// TIA Portal V18 program export: 0 tag tables, 0 data types, 8 data blocks, 19 code blocks (in call order from the OBs), 10 instance data blocks

DATA_BLOCK "settingsShift"   // DB23
{ S7_Optimized_Access := 'TRUE' }
VERSION : 0.1
// stored: AutoNumber false, DBAccessibleFromOPCUA true, DBAccessibleFromWebserver true, IsOnlyStoredInLoadMemory false, IsRetainMemResEnabled true, IsWriteProtectedInAS false, MemoryReserve 1000, RetainMemoryReserve 1000
   VAR RETAIN
      "1" { ExternalVisible := 'False'; S7_SetPoint := 'True'} : "UDT_settingsShift";
      "2" { ExternalVisible := 'False'; S7_SetPoint := 'True'} : "UDT_settingsShift";
      "3" { ExternalVisible := 'False'; S7_SetPoint := 'True'} : "UDT_settingsShift";
   END_VAR
BEGIN
END_DATA_BLOCK

DATA_BLOCK "settingsSirene"   // DB25
{ S7_Optimized_Access := 'TRUE' }
VERSION : 0.1
// stored: AutoNumber false, DBAccessibleFromOPCUA true, DBAccessibleFromWebserver true, IsOnlyStoredInLoadMemory false, IsRetainMemResEnabled true, IsWriteProtectedInAS false, MemoryReserve 100, RetainMemoryReserve 100
   VAR RETAIN
      green { S7_SetPoint := 'True'} : "UDT_settingsSirene";
      yellow { S7_SetPoint := 'True'} : "UDT_settingsSirene";
      red { S7_SetPoint := 'True'} : "UDT_settingsSirene";
   END_VAR
BEGIN
END_DATA_BLOCK

DATA_BLOCK "gDb_AndonBoxConfig"   // DB17
{ S7_Optimized_Access := 'TRUE' }
VERSION : 0.1
// stored: AutoNumber true, DBAccessibleFromOPCUA true, DBAccessibleFromWebserver true, IsOnlyStoredInLoadMemory false, IsRetainMemResEnabled false, IsWriteProtectedInAS false, MemoryReserve 100
   VAR RETAIN
      flashingPeriod : Time := T#200ms;
      EnableAndon1 : Bool := true;
      EnableAndon2 : Bool := true;
      EnableAndon3 : Bool := true;
      EnableAndon4 : Bool := true;
      EnableAndon5 : Bool := true;
      EnableAndon6 : Bool := true;
      EnableAndon7 : Bool := true;
      EnableAndon8 : Bool;
      EnableAndon9 : Bool;
      EnableAndon10 : Bool;
   END_VAR
BEGIN
END_DATA_BLOCK

DATA_BLOCK "gDb_LED_state"   // DB9
{ S7_Optimized_Access := 'TRUE' }
VERSION : 0.1
// stored: AutoNumber true, DBAccessibleFromOPCUA true, DBAccessibleFromWebserver true, IsOnlyStoredInLoadMemory false, IsRetainMemResEnabled false, IsWriteProtectedInAS false, MemoryReserve 100
   VAR RETAIN
      green : Bool;
      yellow : Bool;
      red : Bool;
   END_VAR
BEGIN
END_DATA_BLOCK

DATA_BLOCK "gDb_IO"   // DB20
{ S7_Optimized_Access := 'TRUE' }
VERSION : 0.1
// stored: AutoNumber true, DBAccessibleFromOPCUA true, DBAccessibleFromWebserver true, IsOnlyStoredInLoadMemory false, IsRetainMemResEnabled false, IsWriteProtectedInAS false, MemoryReserve 100
   VAR
      Andon1 : "UDT_andonIO";
      Andon2 : "UDT_andonIO";
      Andon3 : "UDT_andonIO";
      Andon4 : "UDT_andonIO";
      Andon5 : "UDT_andonIO";
      Andon6 : "UDT_andonIO";
      Andon7 : "UDT_andonIO";
      Andon8 : "UDT_andonIO";
      Andon9 : "UDT_andonIO";
      Andon10 : "UDT_andonIO";
      Sirene { S7_SetPoint := 'True'} : "UDT_sireneIO";
      SignalColumn { S7_SetPoint := 'True'} : "UDT_signalColumn";
      NokButton1 { S7_SetPoint := 'True'} : "UDT_nokButtonIO";
      NokButton2 { S7_SetPoint := 'True'} : "UDT_nokButtonIO";
      I_PartProduced { S7_SetPoint := 'True'} : Bool;
   END_VAR
BEGIN
END_DATA_BLOCK

DATA_BLOCK "gdb_nokButton"   // DB14
{ S7_Optimized_Access := 'TRUE' }
VERSION : 0.1
// stored: AutoNumber true, DBAccessibleFromOPCUA true, DBAccessibleFromWebserver true, IsOnlyStoredInLoadMemory false, IsRetainMemResEnabled false, IsWriteProtectedInAS false, MemoryReserve 100
   VAR
      ButtonQue : Int;
      nokPart : Bool;
   END_VAR
BEGIN
END_DATA_BLOCK

DATA_BLOCK "gdb_Sirene"   // DB13
{ S7_Optimized_Access := 'TRUE' }
VERSION : 0.1
// stored: AutoNumber true, DBAccessibleFromOPCUA true, DBAccessibleFromWebserver true, IsOnlyStoredInLoadMemory false, IsRetainMemResEnabled false, IsWriteProtectedInAS false, MemoryReserve 100
   VAR
      greenTrigger : Bool;
      yellowTrigger : Bool;
      redTrigger : Bool;
   END_VAR
BEGIN
END_DATA_BLOCK

DATA_BLOCK "webData"   // DB8
{ S7_Optimized_Access := 'TRUE' }
VERSION : 0.1
// stored: AutoNumber true, DBAccessibleFromOPCUA true, DBAccessibleFromWebserver true, IsOnlyStoredInLoadMemory false, IsRetainMemResEnabled false, IsWriteProtectedInAS false, MemoryReserve 0
   VAR
      lineName { ExternalAccessible := 'False'; ExternalVisible := 'False'; ExternalWritable := 'False'} : WString := WSTRING#'L14';
      andon1Text { ExternalAccessible := 'False'; ExternalVisible := 'False'; ExternalWritable := 'False'} : WString := WSTRING#'Andon1';
      andon2Text { ExternalAccessible := 'False'; ExternalVisible := 'False'; ExternalWritable := 'False'} : WString := WSTRING#'Andon2';
      andon3Text { ExternalAccessible := 'False'; ExternalVisible := 'False'; ExternalWritable := 'False'} : WString := WSTRING#'Andon3';
      andon4Text { ExternalAccessible := 'False'; ExternalVisible := 'False'; ExternalWritable := 'False'} : WString := WSTRING#'Andon4';
      andon5Text { ExternalAccessible := 'False'; ExternalVisible := 'False'; ExternalWritable := 'False'} : WString := WSTRING#'Andon5';
      andon6Text { ExternalAccessible := 'False'; ExternalVisible := 'False'; ExternalWritable := 'False'} : WString := WSTRING#'Andon6';
      andon7Text { ExternalAccessible := 'False'; ExternalVisible := 'False'; ExternalWritable := 'False'} : WString := WSTRING#'Andon7';
      andon8Text { ExternalAccessible := 'False'; ExternalVisible := 'False'; ExternalWritable := 'False'} : WString := WSTRING#'Andon8';
      andon9Text { ExternalAccessible := 'False'; ExternalVisible := 'False'; ExternalWritable := 'False'} : WString := WSTRING#'Andon9';
      andon10Text { ExternalAccessible := 'False'; ExternalVisible := 'False'; ExternalWritable := 'False'} : WString := WSTRING#'Andon10';
      actualValues { ExternalAccessible := 'False'; ExternalVisible := 'False'; ExternalWritable := 'False'} : "UDT_actualValues";
      andon1state { ExternalAccessible := 'False'; ExternalVisible := 'False'; ExternalWritable := 'False'} : Int;
      andon2state { ExternalAccessible := 'False'; ExternalVisible := 'False'; ExternalWritable := 'False'} : Int;
      andon3state { ExternalAccessible := 'False'; ExternalVisible := 'False'; ExternalWritable := 'False'} : Int;
      andon4state { ExternalAccessible := 'False'; ExternalVisible := 'False'; ExternalWritable := 'False'} : Int;
      andon5state { ExternalAccessible := 'False'; ExternalVisible := 'False'; ExternalWritable := 'False'} : Int;
      andon6state { ExternalAccessible := 'False'; ExternalVisible := 'False'; ExternalWritable := 'False'} : Int;
      andon7state { ExternalAccessible := 'False'; ExternalVisible := 'False'; ExternalWritable := 'False'} : Int;
      andon8state { ExternalAccessible := 'False'; ExternalVisible := 'False'; ExternalWritable := 'False'} : Int;
      andon9state { ExternalAccessible := 'False'; ExternalVisible := 'False'; ExternalWritable := 'False'} : Int;
      andon10state { ExternalAccessible := 'False'; ExternalVisible := 'False'; ExternalWritable := 'False'} : Int;
   END_VAR
BEGIN
END_DATA_BLOCK

ORGANIZATION_BLOCK "Main"   // OB1, FBD, ProgramCycle
TITLE = "Main Program Sweep (Cycle)"
{ S7_Optimized_Access := 'TRUE' }
// stored: SetENOAutomatically false
   VAR_INPUT
      Initial_Call : Bool;   // Initial call of this OB
      Remanence : Bool;   // =True, if remanent data are available
   END_VAR
   VAR_TEMP
      RET_VAL : Int;
      locTime : DTL;
   END_VAR
BEGIN

REGION Network 1: Inputs
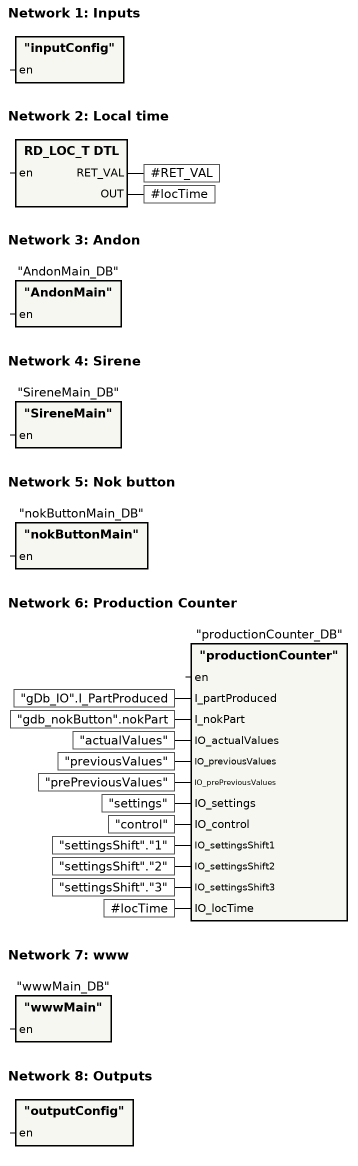
   "inputConfig"();
END_REGION

REGION Network 2: Local time
   #RET_VAL := RD_LOC_T(OUT => #locTime);
END_REGION

REGION Network 3: Andon
   "AndonMain_DB"();   // "AndonMain"
END_REGION

REGION Network 4: Sirene
   "SireneMain_DB"();   // "SireneMain"
END_REGION

REGION Network 5: Nok button
   "nokButtonMain_DB"();   // "nokButtonMain"
END_REGION

REGION Network 6: Production Counter
   "productionCounter_DB"(I_partProduced := "gDb_IO".I_PartProduced,   // "productionCounter"
                          I_nokPart := "gdb_nokButton".nokPart,
                          IO_actualValues := "actualValues",
                          IO_previousValues := "previousValues",
                          IO_prePreviousValues := "prePreviousValues",
                          IO_settings := "settings",
                          IO_control := "control",
                          IO_settingsShift1 := "settingsShift"."1",
                          IO_settingsShift2 := "settingsShift"."2",
                          IO_settingsShift3 := "settingsShift"."3",
                          IO_locTime := #locTime);
END_REGION

REGION Network 7: www
   "wwwMain_DB"();   // "wwwMain"
END_REGION

REGION Network 8: Outputs
   "outputConfig"();
END_REGION
END_ORGANIZATION_BLOCK

FUNCTION "inputConfig" : Void
{ S7_Optimized_Access := 'TRUE' }
VERSION : 0.1

BEGIN
	(*
	//Andon1
	"gDb_IO".Andon1.I_greenBtn := "Andon1_greenBtn";
	"gDb_IO".Andon1.I_yellowBtn := "Andon1_yellowBtn";
	"gDb_IO".Andon1.I_redBtn := "Andon1_redBtn";
	//Andon2
	"gDb_IO".Andon2.I_greenBtn := "Andon2_greenBtn";
	"gDb_IO".Andon2.I_yellowBtn := "Andon2_yellowBtn";
	"gDb_IO".Andon2.I_redBtn := "Andon2_redBtn";
	//Andon7
	"gDb_IO".Andon3.I_greenBtn := "Andon3_greenBtn";
	"gDb_IO".Andon3.I_yellowBtn := "Andon3_yellowBtn";
	"gDb_IO".Andon3.I_redBtn := "Andon3_redBtn";
	//Andon4
	"gDb_IO".Andon4.I_greenBtn := "Andon4_greenBtn";
	"gDb_IO".Andon4.I_yellowBtn := "Andon4_yellowBtn";
	"gDb_IO".Andon4.I_redBtn := "Andon4_redBtn";
	//Andon6
	"gDb_IO".Andon5.I_greenBtn := "Andon5_greenBtn";
	"gDb_IO".Andon5.I_yellowBtn := "Andon5_yellowBtn";
	"gDb_IO".Andon5.I_redBtn := "Andon5_redBtn";
	//Andon6
	"gDb_IO".Andon6.I_greenBtn := "Andon6_greenBtn";
	"gDb_IO".Andon6.I_yellowBtn := "Andon6_yellowBtn";
	"gDb_IO".Andon6.I_redBtn := "Andon6_redBtn";
	//Andon7
	"gDb_IO".Andon7.I_greenBtn := "Andon7_greenBtn";
	"gDb_IO".Andon7.I_yellowBtn := "Andon7_yellowBtn";
	"gDb_IO".Andon7.I_redBtn := "Andon7_redBtn";
	//Andon8
	"gDb_IO".Andon8.I_greenBtn := "Andon8_greenBtn";
	"gDb_IO".Andon8.I_yellowBtn := "Andon8_yellowBtn";
	"gDb_IO".Andon8.I_redBtn := "Andon8_redBtn";
	//Andon9
	"gDb_IO".Andon9.I_greenBtn := "Andon9_greenBtn";
	"gDb_IO".Andon9.I_yellowBtn := "Andon9_yellowBtn";
	"gDb_IO".Andon9.I_redBtn := "Andon9_redBtn";
	*)
END_FUNCTION

FUNCTION_BLOCK "AndonMain"   // FB1, FBD
{ S7_Optimized_Access := 'TRUE' }
VERSION : 0.1
// stored: AutoNumber true, IsIECCheckEnabled false, IsRetainMemResEnabled false, MemoryReserve 100, SetENOAutomatically false, UDAEnableTagReadback false
   VAR
      fpBit_greenTrigger : Bool;
      AndonBoxASi_v2_Instance_8 { S7_SetPoint := 'True'} : "AndonBoxASi";
      AndonBoxASi_v2_Instance_9 { S7_SetPoint := 'True'} : "AndonBoxASi";
      AndonBoxASi_v2_Instance1 { S7_SetPoint := 'True'} : "AndonBoxASi";
      AndonBoxASi_v2_Instance2 { S7_SetPoint := 'True'} : "AndonBoxASi";
      AndonBoxASi_v2_Instance3 { S7_SetPoint := 'True'} : "AndonBoxASi";
      AndonBoxASi_v2_Instance4 { S7_SetPoint := 'True'} : "AndonBoxASi";
      AndonBoxASi_v2_Instance5 { S7_SetPoint := 'True'} : "AndonBoxASi";
      AndonBoxASi_v2_Instance6 { S7_SetPoint := 'True'} : "AndonBoxASi";
      AndonBoxASi_v2_Instance7 { S7_SetPoint := 'True'} : "AndonBoxASi";
      AndonBoxASi_v2_Instance10 { S7_SetPoint := 'True'} : "AndonBoxASi";
   END_VAR
   VAR_TEMP   // added for the SCL form of the ladder/FBD networks
      _w1 : Bool;
      _w2 : Bool;
   END_VAR
BEGIN

REGION Network 1: Green trigger
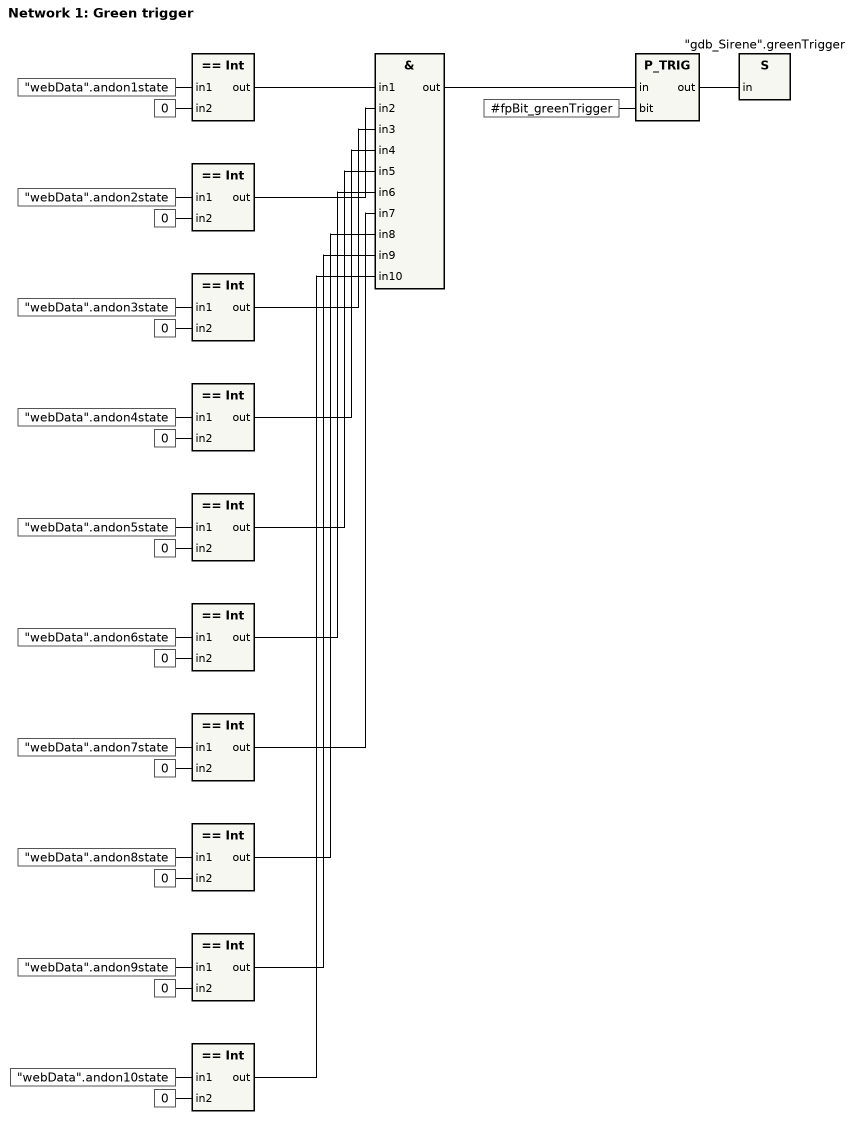
   #_w1 := ("webData".andon1state = 0) AND ("webData".andon2state = 0) AND ("webData".andon3state = 0) AND ("webData".andon4state = 0) AND ("webData".andon5state = 0) AND ("webData".andon6state = 0) AND ("webData".andon7state = 0) AND ("webData".andon8state = 0) AND ("webData".andon9state = 0) AND ("webData".andon10state = 0);
   #_w2 := #_w1 AND NOT #fpBit_greenTrigger;   // rising edge
   #fpBit_greenTrigger := #_w1;
   IF #_w2 THEN "gdb_Sirene".greenTrigger := TRUE; END_IF;
END_REGION

REGION Network 2: Andon1
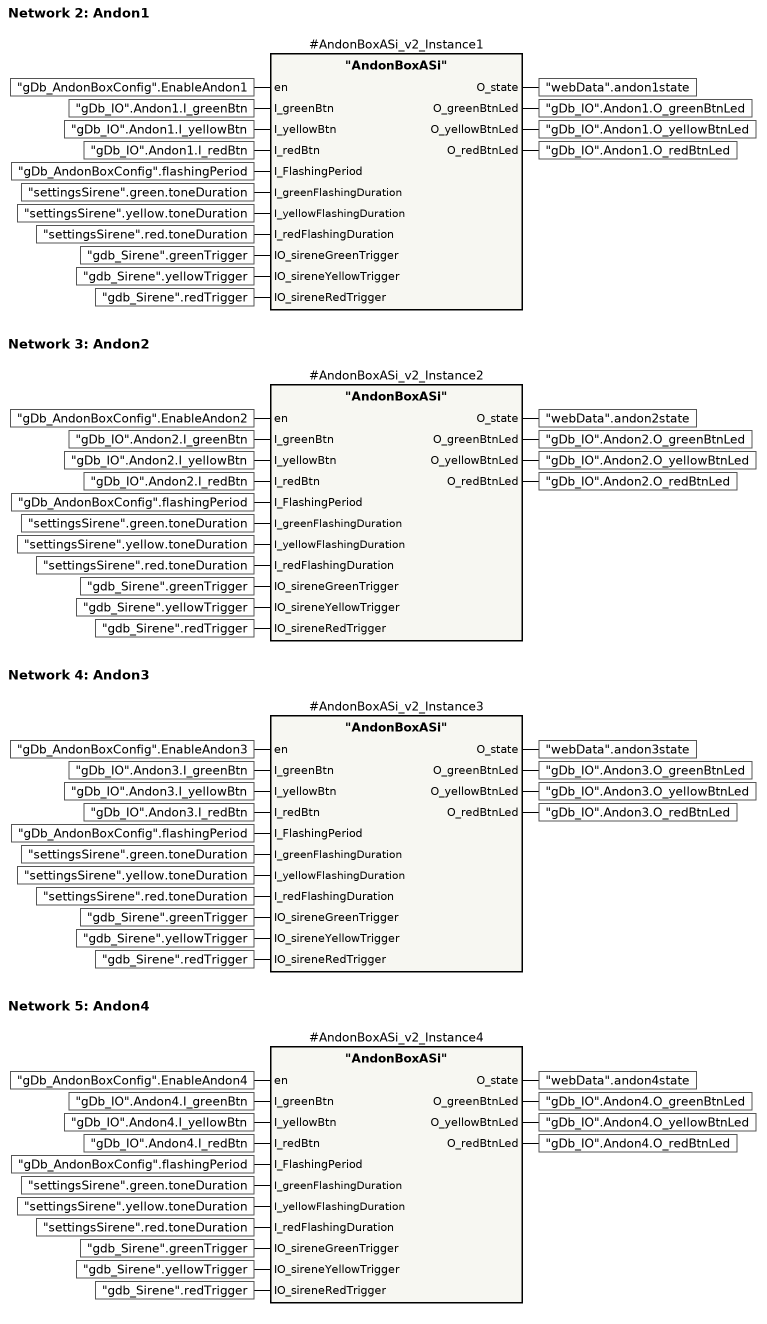
   IF "gDb_AndonBoxConfig".EnableAndon1 THEN
       #AndonBoxASi_v2_Instance1(I_greenBtn := "gDb_IO".Andon1.I_greenBtn,   // "AndonBoxASi"
                               I_yellowBtn := "gDb_IO".Andon1.I_yellowBtn,
                               I_redBtn := "gDb_IO".Andon1.I_redBtn,
                               I_FlashingPeriod := "gDb_AndonBoxConfig".flashingPeriod,
                               I_greenFlashingDuration := "settingsSirene".green.toneDuration,
                               I_yellowFlashingDuration := "settingsSirene".yellow.toneDuration,
                               I_redFlashingDuration := "settingsSirene".red.toneDuration,
                               IO_sireneGreenTrigger := "gdb_Sirene".greenTrigger,
                               IO_sireneYellowTrigger := "gdb_Sirene".yellowTrigger,
                               IO_sireneRedTrigger := "gdb_Sirene".redTrigger,
                               O_state => "webData".andon1state,
                               O_greenBtnLed => "gDb_IO".Andon1.O_greenBtnLed,
                               O_yellowBtnLed => "gDb_IO".Andon1.O_yellowBtnLed,
                               O_redBtnLed => "gDb_IO".Andon1.O_redBtnLed);
   END_IF;
END_REGION

REGION Network 3: Andon2
   IF "gDb_AndonBoxConfig".EnableAndon2 THEN
       #AndonBoxASi_v2_Instance2(I_greenBtn := "gDb_IO".Andon2.I_greenBtn,   // "AndonBoxASi"
                               I_yellowBtn := "gDb_IO".Andon2.I_yellowBtn,
                               I_redBtn := "gDb_IO".Andon2.I_redBtn,
                               I_FlashingPeriod := "gDb_AndonBoxConfig".flashingPeriod,
                               I_greenFlashingDuration := "settingsSirene".green.toneDuration,
                               I_yellowFlashingDuration := "settingsSirene".yellow.toneDuration,
                               I_redFlashingDuration := "settingsSirene".red.toneDuration,
                               IO_sireneGreenTrigger := "gdb_Sirene".greenTrigger,
                               IO_sireneYellowTrigger := "gdb_Sirene".yellowTrigger,
                               IO_sireneRedTrigger := "gdb_Sirene".redTrigger,
                               O_state => "webData".andon2state,
                               O_greenBtnLed => "gDb_IO".Andon2.O_greenBtnLed,
                               O_yellowBtnLed => "gDb_IO".Andon2.O_yellowBtnLed,
                               O_redBtnLed => "gDb_IO".Andon2.O_redBtnLed);
   END_IF;
END_REGION

REGION Network 4: Andon3
   IF "gDb_AndonBoxConfig".EnableAndon3 THEN
       #AndonBoxASi_v2_Instance3(I_greenBtn := "gDb_IO".Andon3.I_greenBtn,   // "AndonBoxASi"
                               I_yellowBtn := "gDb_IO".Andon3.I_yellowBtn,
                               I_redBtn := "gDb_IO".Andon3.I_redBtn,
                               I_FlashingPeriod := "gDb_AndonBoxConfig".flashingPeriod,
                               I_greenFlashingDuration := "settingsSirene".green.toneDuration,
                               I_yellowFlashingDuration := "settingsSirene".yellow.toneDuration,
                               I_redFlashingDuration := "settingsSirene".red.toneDuration,
                               IO_sireneGreenTrigger := "gdb_Sirene".greenTrigger,
                               IO_sireneYellowTrigger := "gdb_Sirene".yellowTrigger,
                               IO_sireneRedTrigger := "gdb_Sirene".redTrigger,
                               O_state => "webData".andon3state,
                               O_greenBtnLed => "gDb_IO".Andon3.O_greenBtnLed,
                               O_yellowBtnLed => "gDb_IO".Andon3.O_yellowBtnLed,
                               O_redBtnLed => "gDb_IO".Andon3.O_redBtnLed);
   END_IF;
END_REGION

REGION Network 5: Andon4
   IF "gDb_AndonBoxConfig".EnableAndon4 THEN
       #AndonBoxASi_v2_Instance4(I_greenBtn := "gDb_IO".Andon4.I_greenBtn,   // "AndonBoxASi"
                               I_yellowBtn := "gDb_IO".Andon4.I_yellowBtn,
                               I_redBtn := "gDb_IO".Andon4.I_redBtn,
                               I_FlashingPeriod := "gDb_AndonBoxConfig".flashingPeriod,
                               I_greenFlashingDuration := "settingsSirene".green.toneDuration,
                               I_yellowFlashingDuration := "settingsSirene".yellow.toneDuration,
                               I_redFlashingDuration := "settingsSirene".red.toneDuration,
                               IO_sireneGreenTrigger := "gdb_Sirene".greenTrigger,
                               IO_sireneYellowTrigger := "gdb_Sirene".yellowTrigger,
                               IO_sireneRedTrigger := "gdb_Sirene".redTrigger,
                               O_state => "webData".andon4state,
                               O_greenBtnLed => "gDb_IO".Andon4.O_greenBtnLed,
                               O_yellowBtnLed => "gDb_IO".Andon4.O_yellowBtnLed,
                               O_redBtnLed => "gDb_IO".Andon4.O_redBtnLed);
   END_IF;
END_REGION

REGION Network 6: Andon5
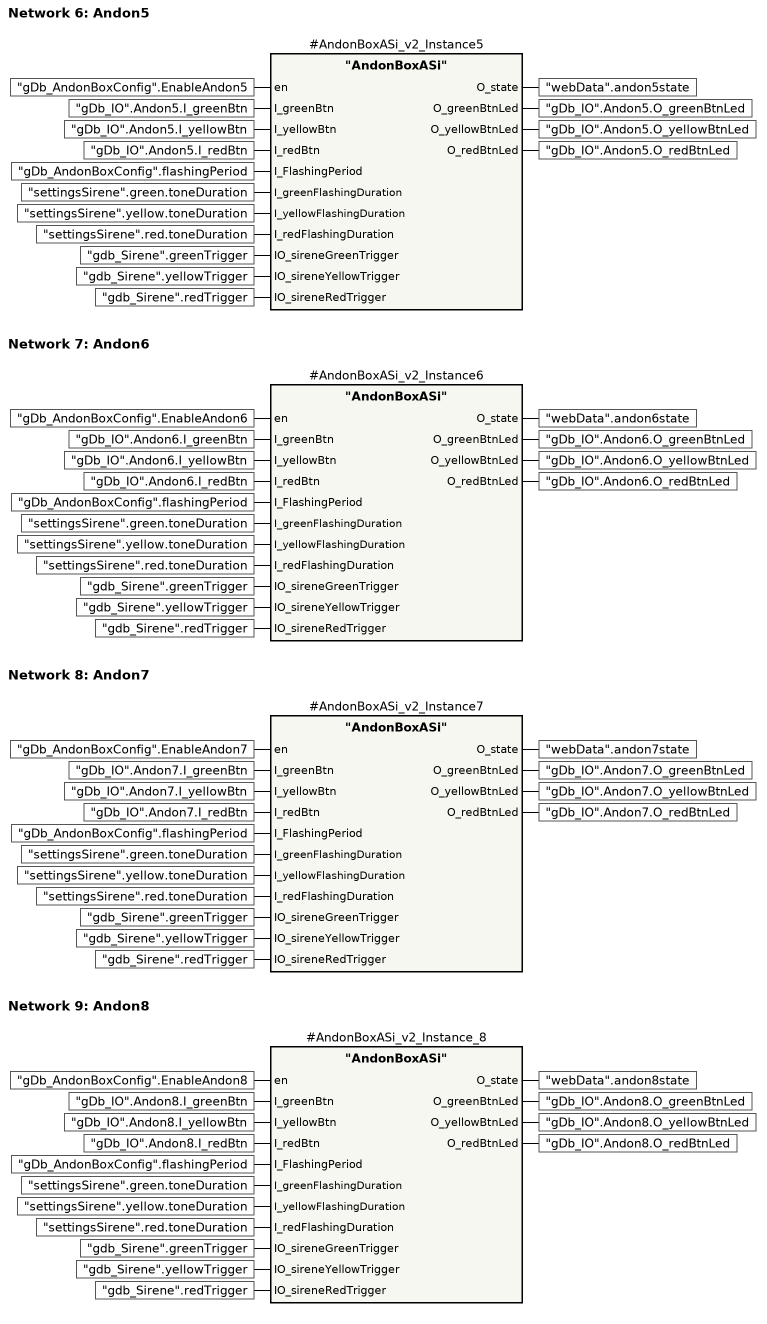
   IF "gDb_AndonBoxConfig".EnableAndon5 THEN
       #AndonBoxASi_v2_Instance5(I_greenBtn := "gDb_IO".Andon5.I_greenBtn,   // "AndonBoxASi"
                               I_yellowBtn := "gDb_IO".Andon5.I_yellowBtn,
                               I_redBtn := "gDb_IO".Andon5.I_redBtn,
                               I_FlashingPeriod := "gDb_AndonBoxConfig".flashingPeriod,
                               I_greenFlashingDuration := "settingsSirene".green.toneDuration,
                               I_yellowFlashingDuration := "settingsSirene".yellow.toneDuration,
                               I_redFlashingDuration := "settingsSirene".red.toneDuration,
                               IO_sireneGreenTrigger := "gdb_Sirene".greenTrigger,
                               IO_sireneYellowTrigger := "gdb_Sirene".yellowTrigger,
                               IO_sireneRedTrigger := "gdb_Sirene".redTrigger,
                               O_state => "webData".andon5state,
                               O_greenBtnLed => "gDb_IO".Andon5.O_greenBtnLed,
                               O_yellowBtnLed => "gDb_IO".Andon5.O_yellowBtnLed,
                               O_redBtnLed => "gDb_IO".Andon5.O_redBtnLed);
   END_IF;
END_REGION

REGION Network 7: Andon6
   IF "gDb_AndonBoxConfig".EnableAndon6 THEN
       #AndonBoxASi_v2_Instance6(I_greenBtn := "gDb_IO".Andon6.I_greenBtn,   // "AndonBoxASi"
                               I_yellowBtn := "gDb_IO".Andon6.I_yellowBtn,
                               I_redBtn := "gDb_IO".Andon6.I_redBtn,
                               I_FlashingPeriod := "gDb_AndonBoxConfig".flashingPeriod,
                               I_greenFlashingDuration := "settingsSirene".green.toneDuration,
                               I_yellowFlashingDuration := "settingsSirene".yellow.toneDuration,
                               I_redFlashingDuration := "settingsSirene".red.toneDuration,
                               IO_sireneGreenTrigger := "gdb_Sirene".greenTrigger,
                               IO_sireneYellowTrigger := "gdb_Sirene".yellowTrigger,
                               IO_sireneRedTrigger := "gdb_Sirene".redTrigger,
                               O_state => "webData".andon6state,
                               O_greenBtnLed => "gDb_IO".Andon6.O_greenBtnLed,
                               O_yellowBtnLed => "gDb_IO".Andon6.O_yellowBtnLed,
                               O_redBtnLed => "gDb_IO".Andon6.O_redBtnLed);
   END_IF;
END_REGION

REGION Network 8: Andon7
   IF "gDb_AndonBoxConfig".EnableAndon7 THEN
       #AndonBoxASi_v2_Instance7(I_greenBtn := "gDb_IO".Andon7.I_greenBtn,   // "AndonBoxASi"
                               I_yellowBtn := "gDb_IO".Andon7.I_yellowBtn,
                               I_redBtn := "gDb_IO".Andon7.I_redBtn,
                               I_FlashingPeriod := "gDb_AndonBoxConfig".flashingPeriod,
                               I_greenFlashingDuration := "settingsSirene".green.toneDuration,
                               I_yellowFlashingDuration := "settingsSirene".yellow.toneDuration,
                               I_redFlashingDuration := "settingsSirene".red.toneDuration,
                               IO_sireneGreenTrigger := "gdb_Sirene".greenTrigger,
                               IO_sireneYellowTrigger := "gdb_Sirene".yellowTrigger,
                               IO_sireneRedTrigger := "gdb_Sirene".redTrigger,
                               O_state => "webData".andon7state,
                               O_greenBtnLed => "gDb_IO".Andon7.O_greenBtnLed,
                               O_yellowBtnLed => "gDb_IO".Andon7.O_yellowBtnLed,
                               O_redBtnLed => "gDb_IO".Andon7.O_redBtnLed);
   END_IF;
END_REGION

REGION Network 9: Andon8
   IF "gDb_AndonBoxConfig".EnableAndon8 THEN
       #AndonBoxASi_v2_Instance_8(I_greenBtn := "gDb_IO".Andon8.I_greenBtn,   // "AndonBoxASi"
                               I_yellowBtn := "gDb_IO".Andon8.I_yellowBtn,
                               I_redBtn := "gDb_IO".Andon8.I_redBtn,
                               I_FlashingPeriod := "gDb_AndonBoxConfig".flashingPeriod,
                               I_greenFlashingDuration := "settingsSirene".green.toneDuration,
                               I_yellowFlashingDuration := "settingsSirene".yellow.toneDuration,
                               I_redFlashingDuration := "settingsSirene".red.toneDuration,
                               IO_sireneGreenTrigger := "gdb_Sirene".greenTrigger,
                               IO_sireneYellowTrigger := "gdb_Sirene".yellowTrigger,
                               IO_sireneRedTrigger := "gdb_Sirene".redTrigger,
                               O_state => "webData".andon8state,
                               O_greenBtnLed => "gDb_IO".Andon8.O_greenBtnLed,
                               O_yellowBtnLed => "gDb_IO".Andon8.O_yellowBtnLed,
                               O_redBtnLed => "gDb_IO".Andon8.O_redBtnLed);
   END_IF;
END_REGION

REGION Network 10: Andon9
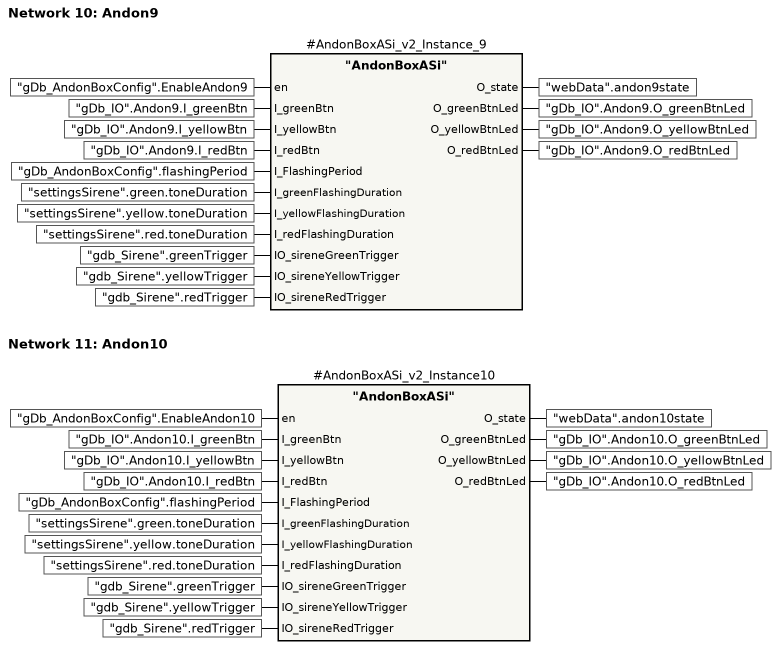
   IF "gDb_AndonBoxConfig".EnableAndon9 THEN
       #AndonBoxASi_v2_Instance_9(I_greenBtn := "gDb_IO".Andon9.I_greenBtn,   // "AndonBoxASi"
                               I_yellowBtn := "gDb_IO".Andon9.I_yellowBtn,
                               I_redBtn := "gDb_IO".Andon9.I_redBtn,
                               I_FlashingPeriod := "gDb_AndonBoxConfig".flashingPeriod,
                               I_greenFlashingDuration := "settingsSirene".green.toneDuration,
                               I_yellowFlashingDuration := "settingsSirene".yellow.toneDuration,
                               I_redFlashingDuration := "settingsSirene".red.toneDuration,
                               IO_sireneGreenTrigger := "gdb_Sirene".greenTrigger,
                               IO_sireneYellowTrigger := "gdb_Sirene".yellowTrigger,
                               IO_sireneRedTrigger := "gdb_Sirene".redTrigger,
                               O_state => "webData".andon9state,
                               O_greenBtnLed => "gDb_IO".Andon9.O_greenBtnLed,
                               O_yellowBtnLed => "gDb_IO".Andon9.O_yellowBtnLed,
                               O_redBtnLed => "gDb_IO".Andon9.O_redBtnLed);
   END_IF;
END_REGION

REGION Network 11: Andon10
   IF "gDb_AndonBoxConfig".EnableAndon10 THEN
       #AndonBoxASi_v2_Instance10(I_greenBtn := "gDb_IO".Andon10.I_greenBtn,   // "AndonBoxASi"
                               I_yellowBtn := "gDb_IO".Andon10.I_yellowBtn,
                               I_redBtn := "gDb_IO".Andon10.I_redBtn,
                               I_FlashingPeriod := "gDb_AndonBoxConfig".flashingPeriod,
                               I_greenFlashingDuration := "settingsSirene".green.toneDuration,
                               I_yellowFlashingDuration := "settingsSirene".yellow.toneDuration,
                               I_redFlashingDuration := "settingsSirene".red.toneDuration,
                               IO_sireneGreenTrigger := "gdb_Sirene".greenTrigger,
                               IO_sireneYellowTrigger := "gdb_Sirene".yellowTrigger,
                               IO_sireneRedTrigger := "gdb_Sirene".redTrigger,
                               O_state => "webData".andon10state,
                               O_greenBtnLed => "gDb_IO".Andon10.O_greenBtnLed,
                               O_yellowBtnLed => "gDb_IO".Andon10.O_yellowBtnLed,
                               O_redBtnLed => "gDb_IO".Andon10.O_redBtnLed);
   END_IF;
END_REGION

REGION Network 12: Semafor red
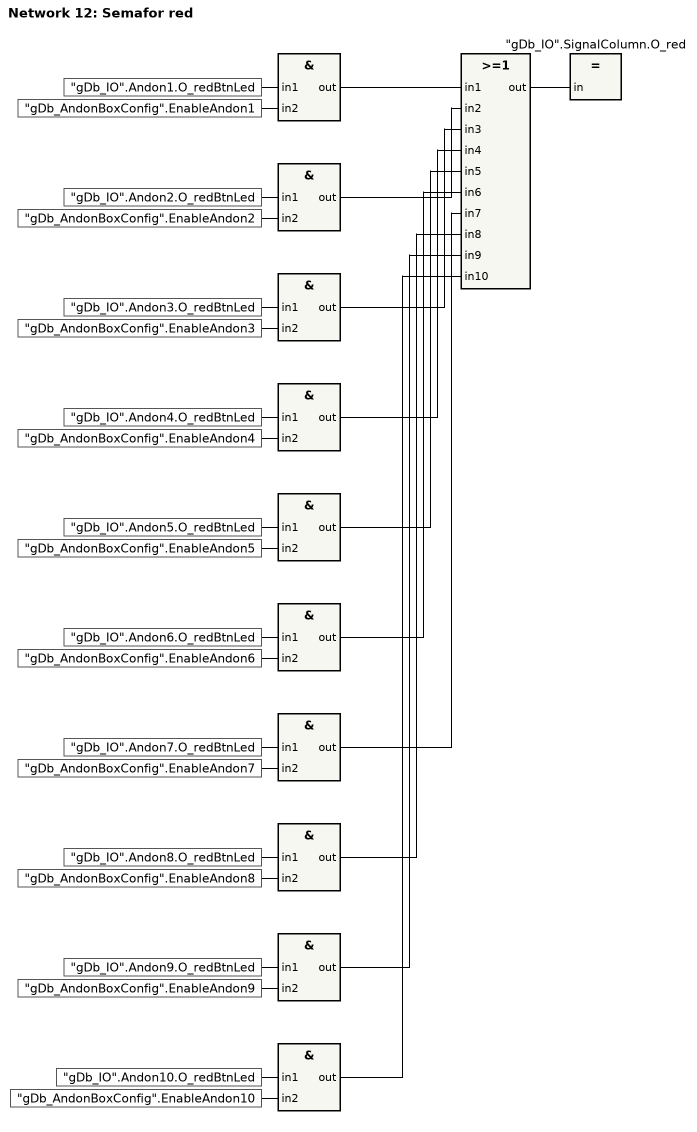
   "gDb_IO".SignalColumn.O_red := ("gDb_IO".Andon1.O_redBtnLed AND "gDb_AndonBoxConfig".EnableAndon1) OR ("gDb_IO".Andon2.O_redBtnLed AND "gDb_AndonBoxConfig".EnableAndon2) OR ("gDb_IO".Andon3.O_redBtnLed AND "gDb_AndonBoxConfig".EnableAndon3) OR ("gDb_IO".Andon4.O_redBtnLed AND "gDb_AndonBoxConfig".EnableAndon4) OR ("gDb_IO".Andon5.O_redBtnLed AND "gDb_AndonBoxConfig".EnableAndon5) OR ("gDb_IO".Andon6.O_redBtnLed AND "gDb_AndonBoxConfig".EnableAndon6) OR ("gDb_IO".Andon7.O_redBtnLed AND "gDb_AndonBoxConfig".EnableAndon7) OR ("gDb_IO".Andon8.O_redBtnLed AND "gDb_AndonBoxConfig".EnableAndon8) OR ("gDb_IO".Andon9.O_redBtnLed AND "gDb_AndonBoxConfig".EnableAndon9) OR ("gDb_IO".Andon10.O_redBtnLed AND "gDb_AndonBoxConfig".EnableAndon10);
END_REGION

REGION Network 13: Semafor yellow
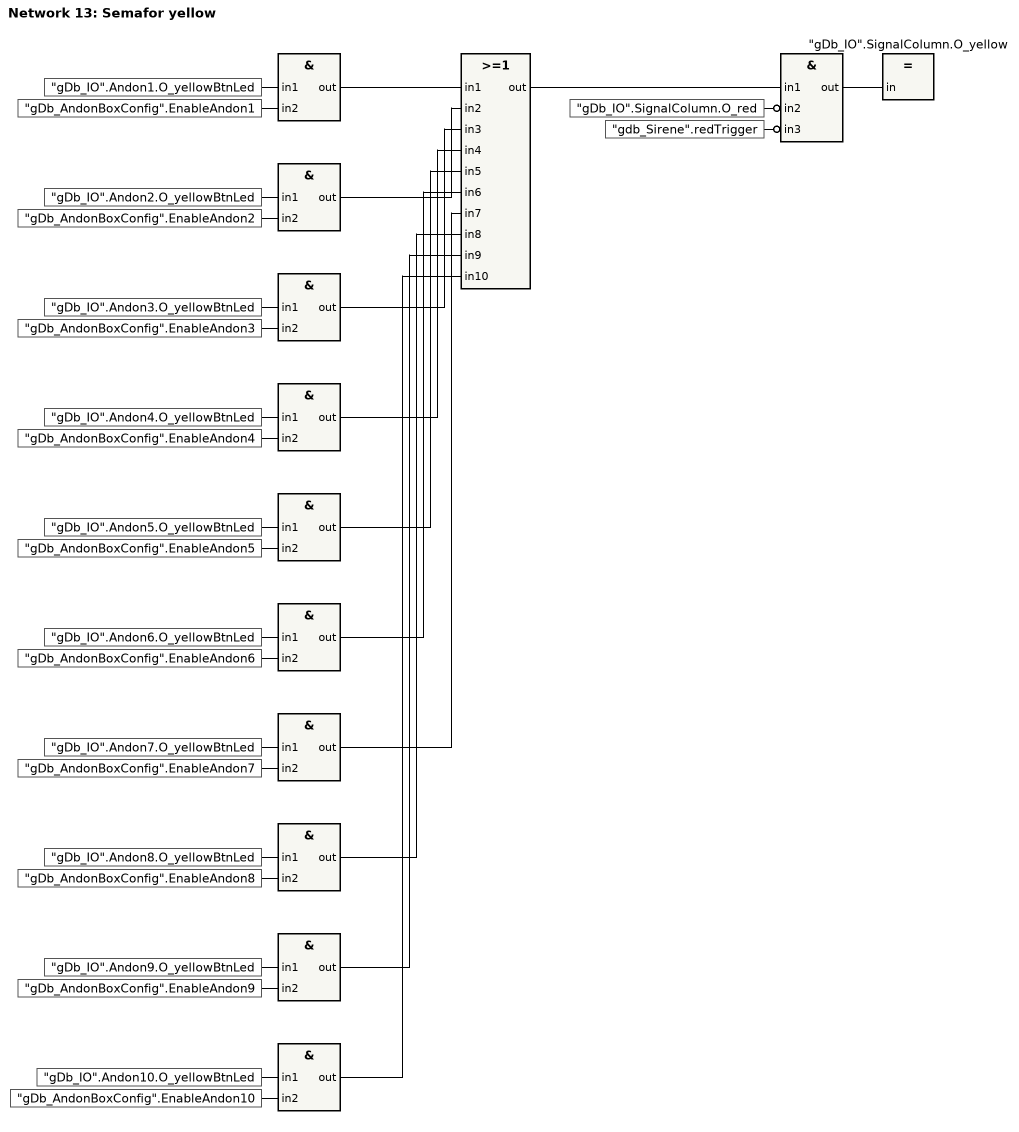
   "gDb_IO".SignalColumn.O_yellow := (("gDb_IO".Andon1.O_yellowBtnLed AND "gDb_AndonBoxConfig".EnableAndon1) OR ("gDb_IO".Andon2.O_yellowBtnLed AND "gDb_AndonBoxConfig".EnableAndon2) OR ("gDb_IO".Andon3.O_yellowBtnLed AND "gDb_AndonBoxConfig".EnableAndon3) OR ("gDb_IO".Andon4.O_yellowBtnLed AND "gDb_AndonBoxConfig".EnableAndon4) OR ("gDb_IO".Andon5.O_yellowBtnLed AND "gDb_AndonBoxConfig".EnableAndon5) OR ("gDb_IO".Andon6.O_yellowBtnLed AND "gDb_AndonBoxConfig".EnableAndon6) OR ("gDb_IO".Andon7.O_yellowBtnLed AND "gDb_AndonBoxConfig".EnableAndon7) OR ("gDb_IO".Andon8.O_yellowBtnLed AND "gDb_AndonBoxConfig".EnableAndon8) OR ("gDb_IO".Andon9.O_yellowBtnLed AND "gDb_AndonBoxConfig".EnableAndon9) OR ("gDb_IO".Andon10.O_yellowBtnLed AND "gDb_AndonBoxConfig".EnableAndon10)) AND NOT "gDb_IO".SignalColumn.O_red AND NOT "gdb_Sirene".redTrigger;
END_REGION

REGION Network 14: Semafor green
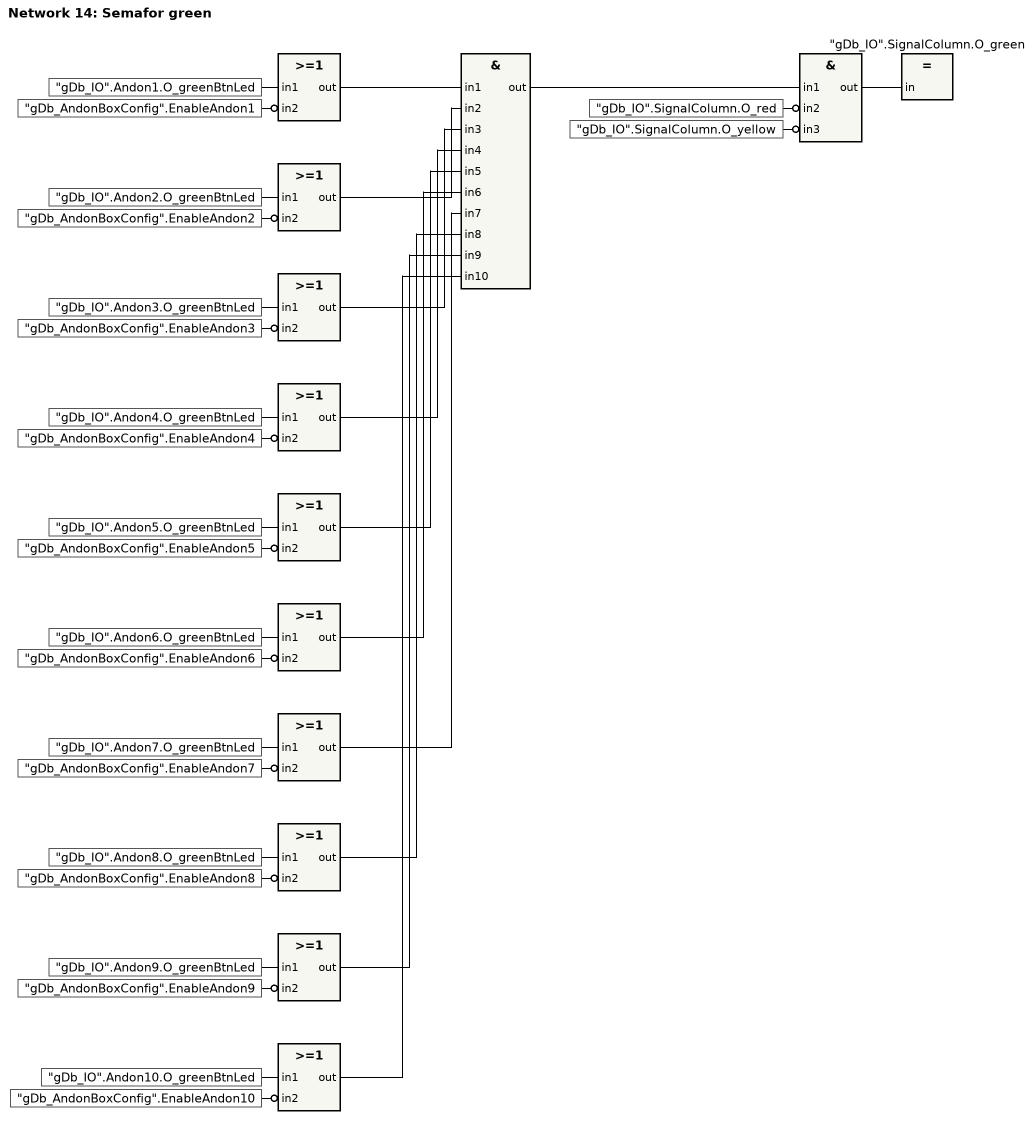
   "gDb_IO".SignalColumn.O_green := ("gDb_IO".Andon1.O_greenBtnLed OR NOT "gDb_AndonBoxConfig".EnableAndon1) AND ("gDb_IO".Andon2.O_greenBtnLed OR NOT "gDb_AndonBoxConfig".EnableAndon2) AND ("gDb_IO".Andon3.O_greenBtnLed OR NOT "gDb_AndonBoxConfig".EnableAndon3) AND ("gDb_IO".Andon4.O_greenBtnLed OR NOT "gDb_AndonBoxConfig".EnableAndon4) AND ("gDb_IO".Andon5.O_greenBtnLed OR NOT "gDb_AndonBoxConfig".EnableAndon5) AND ("gDb_IO".Andon6.O_greenBtnLed OR NOT "gDb_AndonBoxConfig".EnableAndon6) AND ("gDb_IO".Andon7.O_greenBtnLed OR NOT "gDb_AndonBoxConfig".EnableAndon7) AND ("gDb_IO".Andon8.O_greenBtnLed OR NOT "gDb_AndonBoxConfig".EnableAndon8) AND ("gDb_IO".Andon9.O_greenBtnLed OR NOT "gDb_AndonBoxConfig".EnableAndon9) AND ("gDb_IO".Andon10.O_greenBtnLed OR NOT "gDb_AndonBoxConfig".EnableAndon10) AND NOT "gDb_IO".SignalColumn.O_red AND NOT "gDb_IO".SignalColumn.O_yellow;
END_REGION
END_FUNCTION_BLOCK

FUNCTION_BLOCK "AndonBoxASi"   // FB13, FBD
{ S7_Optimized_Access := 'TRUE' }
VERSION : 0.1
// stored: AutoNumber true, IsIECCheckEnabled false, IsRetainMemResEnabled false, MemoryReserve 100, SetENOAutomatically false, UDAEnableTagReadback false
   VAR_INPUT
      I_greenBtn { ExternalAccessible := 'False'; ExternalVisible := 'False'; ExternalWritable := 'False'} : Bool;
      I_yellowBtn { ExternalAccessible := 'False'; ExternalVisible := 'False'; ExternalWritable := 'False'} : Bool;
      I_redBtn { ExternalAccessible := 'False'; ExternalVisible := 'False'; ExternalWritable := 'False'} : Bool;
      I_FlashingPeriod { ExternalAccessible := 'False'; ExternalVisible := 'False'; ExternalWritable := 'False'} : Time;
      I_greenFlashingDuration { ExternalAccessible := 'False'; ExternalVisible := 'False'; ExternalWritable := 'False'} : Time;
      I_yellowFlashingDuration { ExternalAccessible := 'False'; ExternalVisible := 'False'; ExternalWritable := 'False'} : Time;
      I_redFlashingDuration { ExternalAccessible := 'False'; ExternalVisible := 'False'; ExternalWritable := 'False'} : Time;
   END_VAR
   VAR_OUTPUT
      O_state { ExternalAccessible := 'False'; ExternalVisible := 'False'; ExternalWritable := 'False'} : Int;
      O_greenBtnLed { ExternalAccessible := 'False'; ExternalVisible := 'False'; ExternalWritable := 'False'} : Bool;
      O_yellowBtnLed { ExternalAccessible := 'False'; ExternalVisible := 'False'; ExternalWritable := 'False'} : Bool;
      O_redBtnLed { ExternalAccessible := 'False'; ExternalVisible := 'False'; ExternalWritable := 'False'} : Bool;
   END_VAR
   VAR_IN_OUT
      IO_sireneGreenTrigger { ExternalAccessible := 'False'; ExternalVisible := 'False'; ExternalWritable := 'False'} : Bool;
      IO_sireneYellowTrigger { ExternalAccessible := 'False'; ExternalVisible := 'False'; ExternalWritable := 'False'} : Bool;
      IO_sireneRedTrigger { ExternalAccessible := 'False'; ExternalVisible := 'False'; ExternalWritable := 'False'} : Bool;
   END_VAR
   VAR
      fpBit_greenBtn { ExternalAccessible := 'False'; ExternalVisible := 'False'; ExternalWritable := 'False'} : Bool;
      fpBit_yellowBtn { ExternalAccessible := 'False'; ExternalVisible := 'False'; ExternalWritable := 'False'} : Bool;
      fpBit_redBtn { ExternalAccessible := 'False'; ExternalVisible := 'False'; ExternalWritable := 'False'} : Bool;
   END_VAR
   VAR RETAIN
      memState { ExternalAccessible := 'False'; ExternalVisible := 'False'; ExternalWritable := 'False'} : Int;
   END_VAR
   VAR
      IEC_Timer_0_Instance { ExternalAccessible := 'False'; ExternalVisible := 'False'; ExternalWritable := 'False'; S7_SetPoint := 'True'} : TP_TIME;
      BtnLedAppearance_Instance { ExternalAccessible := 'False'; ExternalVisible := 'False'; ExternalWritable := 'False'; S7_SetPoint := 'True'} : "BtnLedAppearance";
      BtnLedAppearance_Instance_1 { ExternalAccessible := 'False'; ExternalVisible := 'False'; ExternalWritable := 'False'; S7_SetPoint := 'True'} : "BtnLedAppearance";
      BtnLedAppearance_Instance_2 { ExternalAccessible := 'False'; ExternalVisible := 'False'; ExternalWritable := 'False'; S7_SetPoint := 'True'} : "BtnLedAppearance";
   END_VAR
   VAR_TEMP
      T_fpGreen : Bool;
      T_fpYellow : Bool;
      T_fpRed : Bool;
   END_VAR
   VAR_TEMP   // added for the SCL form of the ladder/FBD networks
      _w1 : Bool;
   END_VAR
BEGIN

REGION Network 1: positive edge green button
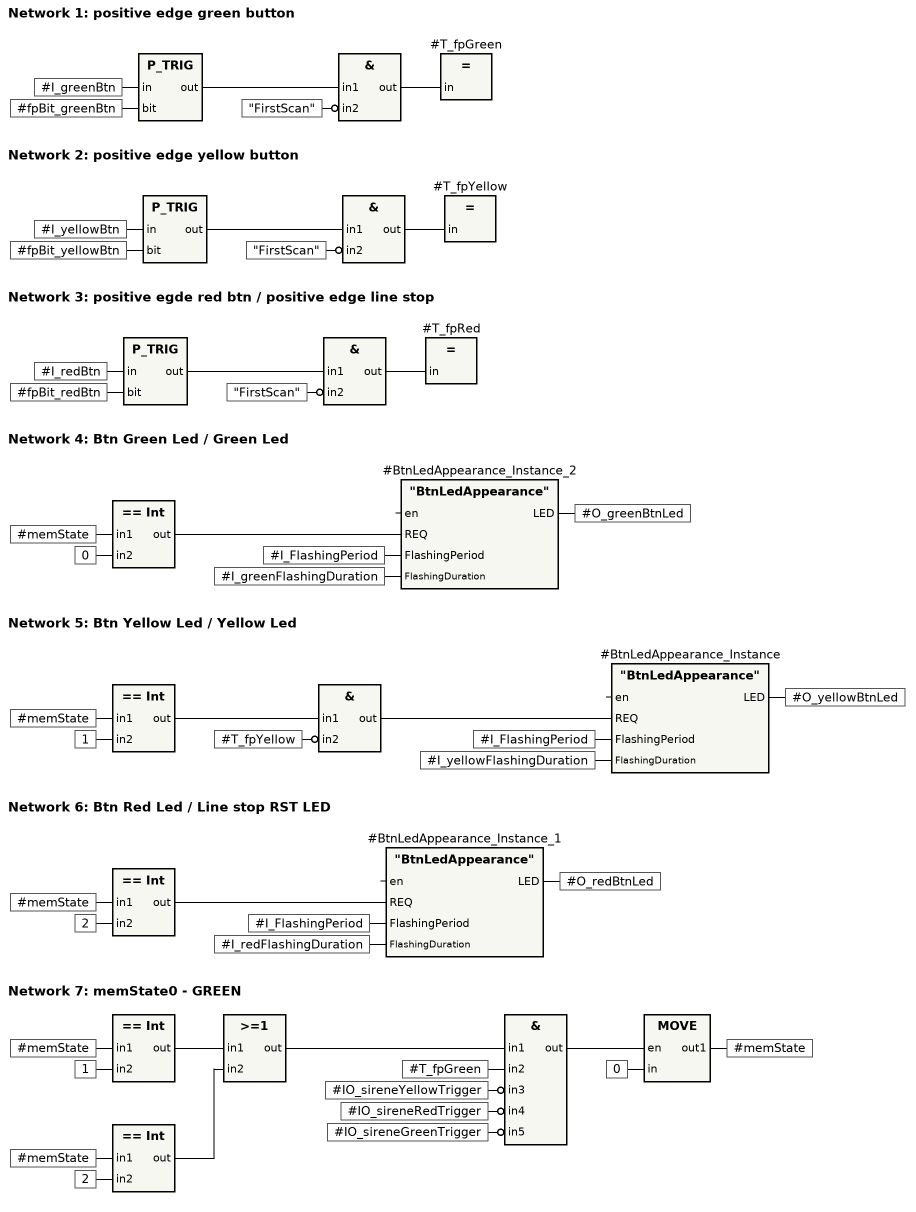
   #_w1 := #I_greenBtn AND NOT #fpBit_greenBtn;   // rising edge
   #fpBit_greenBtn := #I_greenBtn;
   #T_fpGreen := #_w1 AND NOT "FirstScan";
END_REGION

REGION Network 2: positive edge yellow button
   #_w1 := #I_yellowBtn AND NOT #fpBit_yellowBtn;   // rising edge
   #fpBit_yellowBtn := #I_yellowBtn;
   #T_fpYellow := #_w1 AND NOT "FirstScan";
END_REGION

REGION Network 3: positive egde red btn / positive edge line stop
   #_w1 := #I_redBtn AND NOT #fpBit_redBtn;   // rising edge
   #fpBit_redBtn := #I_redBtn;
   #T_fpRed := #_w1 AND NOT "FirstScan";
END_REGION

REGION Network 4: Btn Green Led / Green Led
   #BtnLedAppearance_Instance_2(REQ := #memState = 0,   // "BtnLedAppearance"
                           FlashingPeriod := #I_FlashingPeriod,
                           FlashingDuration := #I_greenFlashingDuration,
                           LED => #O_greenBtnLed);
END_REGION

REGION Network 5: Btn Yellow Led / Yellow Led
   #BtnLedAppearance_Instance(REQ := (#memState = 1) AND NOT #T_fpYellow,   // "BtnLedAppearance"
                           FlashingPeriod := #I_FlashingPeriod,
                           FlashingDuration := #I_yellowFlashingDuration,
                           LED => #O_yellowBtnLed);
END_REGION

REGION Network 6: Btn Red Led / Line stop RST LED
   #BtnLedAppearance_Instance_1(REQ := #memState = 2,   // "BtnLedAppearance"
                           FlashingPeriod := #I_FlashingPeriod,
                           FlashingDuration := #I_redFlashingDuration,
                           LED => #O_redBtnLed);
END_REGION

REGION Network 7: memState0 - GREEN
   IF ((#memState = 1) OR (#memState = 2)) AND #T_fpGreen AND NOT #IO_sireneYellowTrigger AND NOT #IO_sireneRedTrigger AND NOT #IO_sireneGreenTrigger THEN
       #memState := 0;
   END_IF;
END_REGION

REGION Network 8: memState1 - YELLOW / Yellow button / State1
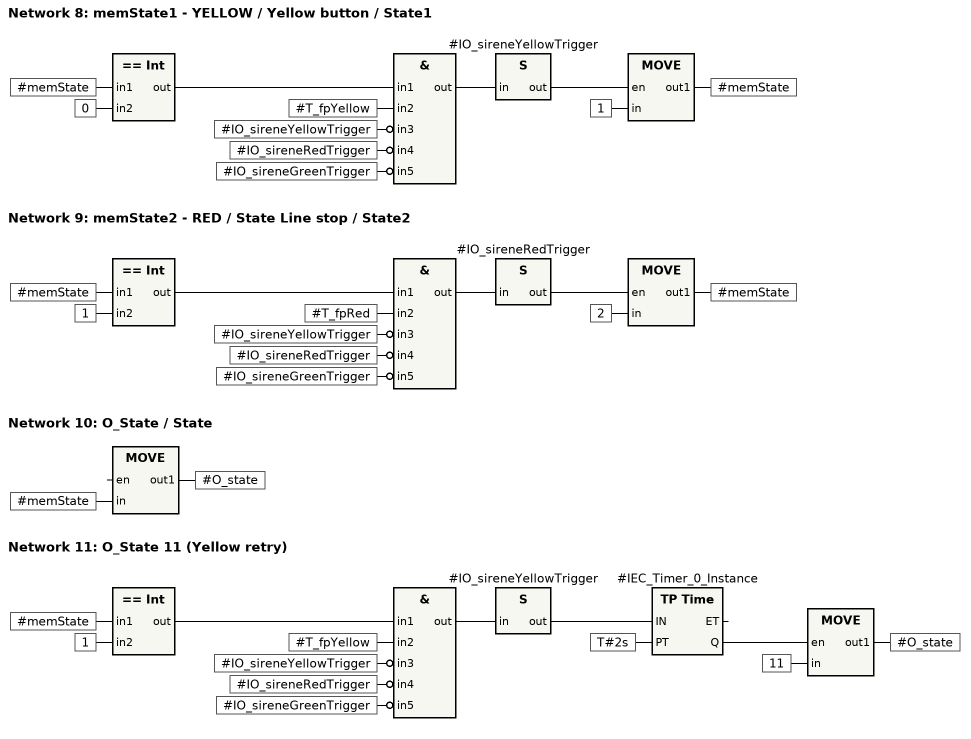
   #_w1 := (#memState = 0) AND #T_fpYellow AND NOT #IO_sireneYellowTrigger AND NOT #IO_sireneRedTrigger AND NOT #IO_sireneGreenTrigger;
   IF #_w1 THEN
       #IO_sireneYellowTrigger := TRUE;
       #memState := 1;
   END_IF;
END_REGION

REGION Network 9: memState2 - RED / State Line stop / State2
   #_w1 := (#memState = 1) AND #T_fpRed AND NOT #IO_sireneYellowTrigger AND NOT #IO_sireneRedTrigger AND NOT #IO_sireneGreenTrigger;
   IF #_w1 THEN
       #IO_sireneRedTrigger := TRUE;
       #memState := 2;
   END_IF;
END_REGION

REGION Network 10: O_State / State
   #O_state := #memState;
END_REGION

REGION Network 11: O_State 11 (Yellow retry)
   #_w1 := (#memState = 1) AND #T_fpYellow AND NOT #IO_sireneYellowTrigger AND NOT #IO_sireneRedTrigger AND NOT #IO_sireneGreenTrigger;
   IF #_w1 THEN #IO_sireneYellowTrigger := TRUE; END_IF;
   #IEC_Timer_0_Instance(IN := #_w1, PT := T#2s);   // TP
   IF #IEC_Timer_0_Instance.Q THEN #O_state := 11; END_IF;
END_REGION
END_FUNCTION_BLOCK

FUNCTION_BLOCK "BtnLedAppearance"
{ S7_Optimized_Access := 'TRUE' }
VERSION : 0.1
   VAR_INPUT 
      REQ : Bool;
      FlashingPeriod : Time;
      FlashingDuration : Time;
   END_VAR

   VAR_OUTPUT 
      LED : Bool;
   END_VAR

   VAR 
      IEC_Timer_ON {InstructionName := 'TON_TIME'; LibVersion := '1.0'} : TON_TIME;
      IEC_Timer_OFF {InstructionName := 'TON_TIME'; LibVersion := '1.0'} : TON_TIME;
      IEC_Timer_TONE_ELAPSED {InstructionName := 'TON_TIME'; LibVersion := '1.0'} : TON_TIME;
   END_VAR


BEGIN
	#IEC_Timer_ON(IN := #REQ AND NOT #IEC_Timer_OFF.Q,
	              PT := #FlashingPeriod);
	
	#IEC_Timer_OFF(IN := #REQ AND #IEC_Timer_ON.Q AND NOT #IEC_Timer_OFF.Q,
	               PT := #FlashingPeriod);
	
	
	#IEC_Timer_TONE_ELAPSED(IN:=#REQ,
	                        PT:=#FlashingDuration);
	
	
	#LED := #IEC_Timer_ON.Q OR #IEC_Timer_TONE_ELAPSED.Q ;
	
END_FUNCTION_BLOCK

FUNCTION_BLOCK "SireneMain"   // FB6, FBD
{ S7_Optimized_Access := 'TRUE' }
VERSION : 0.1
// stored: AutoNumber true, IsIECCheckEnabled false, IsRetainMemResEnabled false, MemoryReserve 100, SetENOAutomatically false, UDAEnableTagReadback false
   VAR
      sirene_Instance { S7_SetPoint := 'True'} : "sirene_v2";
   END_VAR
BEGIN

REGION Network 2: Trigger
END_REGION

REGION Network 3
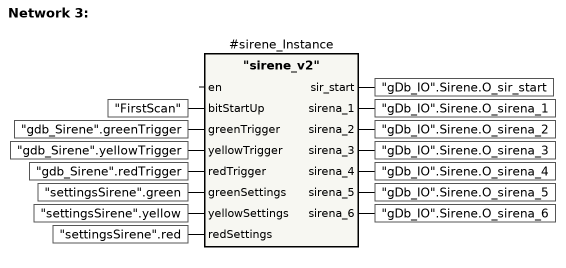
   #sirene_Instance(bitStartUp := "FirstScan",   // "sirene_v2"
                    greenTrigger := "gdb_Sirene".greenTrigger,
                    yellowTrigger := "gdb_Sirene".yellowTrigger,
                    redTrigger := "gdb_Sirene".redTrigger,
                    greenSettings := "settingsSirene".green,
                    yellowSettings := "settingsSirene".yellow,
                    redSettings := "settingsSirene".red,
                    sir_start => "gDb_IO".Sirene.O_sir_start,
                    sirena_1 => "gDb_IO".Sirene.O_sirena_1,
                    sirena_2 => "gDb_IO".Sirene.O_sirena_2,
                    sirena_3 => "gDb_IO".Sirene.O_sirena_3,
                    sirena_4 => "gDb_IO".Sirene.O_sirena_4,
                    sirena_5 => "gDb_IO".Sirene.O_sirena_5,
                    sirena_6 => "gDb_IO".Sirene.O_sirena_6);
END_REGION
END_FUNCTION_BLOCK

FUNCTION_BLOCK "sirene_v2"   // FB7, FBD
{ S7_Optimized_Access := 'TRUE' }
VERSION : 0.1
// stored: AutoNumber true, IsIECCheckEnabled false, IsRetainMemResEnabled false, MemoryReserve 100, SetENOAutomatically false, UDAEnableTagReadback false
   VAR_INPUT
      bitStartUp : Bool;
   END_VAR
   VAR_OUTPUT
      sir_start : Bool;
      sirena_1 : Bool;
      sirena_2 : Bool;
      sirena_3 : Bool;
      sirena_4 : Bool;
      sirena_5 : Bool;
      sirena_6 : Bool;
   END_VAR
   VAR_IN_OUT
      greenTrigger : Bool;
      yellowTrigger : Bool;
      redTrigger : Bool;
      greenSettings : "UDT_settingsSirene";
      yellowSettings : "UDT_settingsSirene";
      redSettings : "UDT_settingsSirene";
   END_VAR
   VAR
      "step" : Int;
      fpBit_green : Bool;
      fpBit_yellow : Bool;
      fpBit_red : Bool;
      fpBit_greenTest : Bool;
      fpBit_yellowTest : Bool;
      fpBit_redTest : Bool;
      IEC_Timer_step1 { S7_SetPoint := 'True'} : IEC_TIMER;
      toneSelect : Int;
      toneDuration : Time;
      IEC_Timer_toneDuration { S7_SetPoint := 'True'} : IEC_TIMER;
      IEC_Timer_step2 { S7_SetPoint := 'True'} : IEC_TIMER;
      sirenaArray { ExternalAccessible := 'False'; ExternalVisible := 'False'; ExternalWritable := 'False'} : Array[0..15] of Bool;
   END_VAR
   VAR_TEMP   // added for the SCL form of the ladder/FBD networks
      _w1 : Bool;
      _w2 : Bool;
      _w3 : Bool;
      _w4 : Bool;
      _w5 : Bool;
      _w6 : Bool;
      _w7 : Bool;
      _w8 : Bool;
      _w9 : Bool;
      _w10 : Bool;
      _w11 : Bool;
      _w12 : Bool;
   END_VAR
BEGIN

REGION Network 2
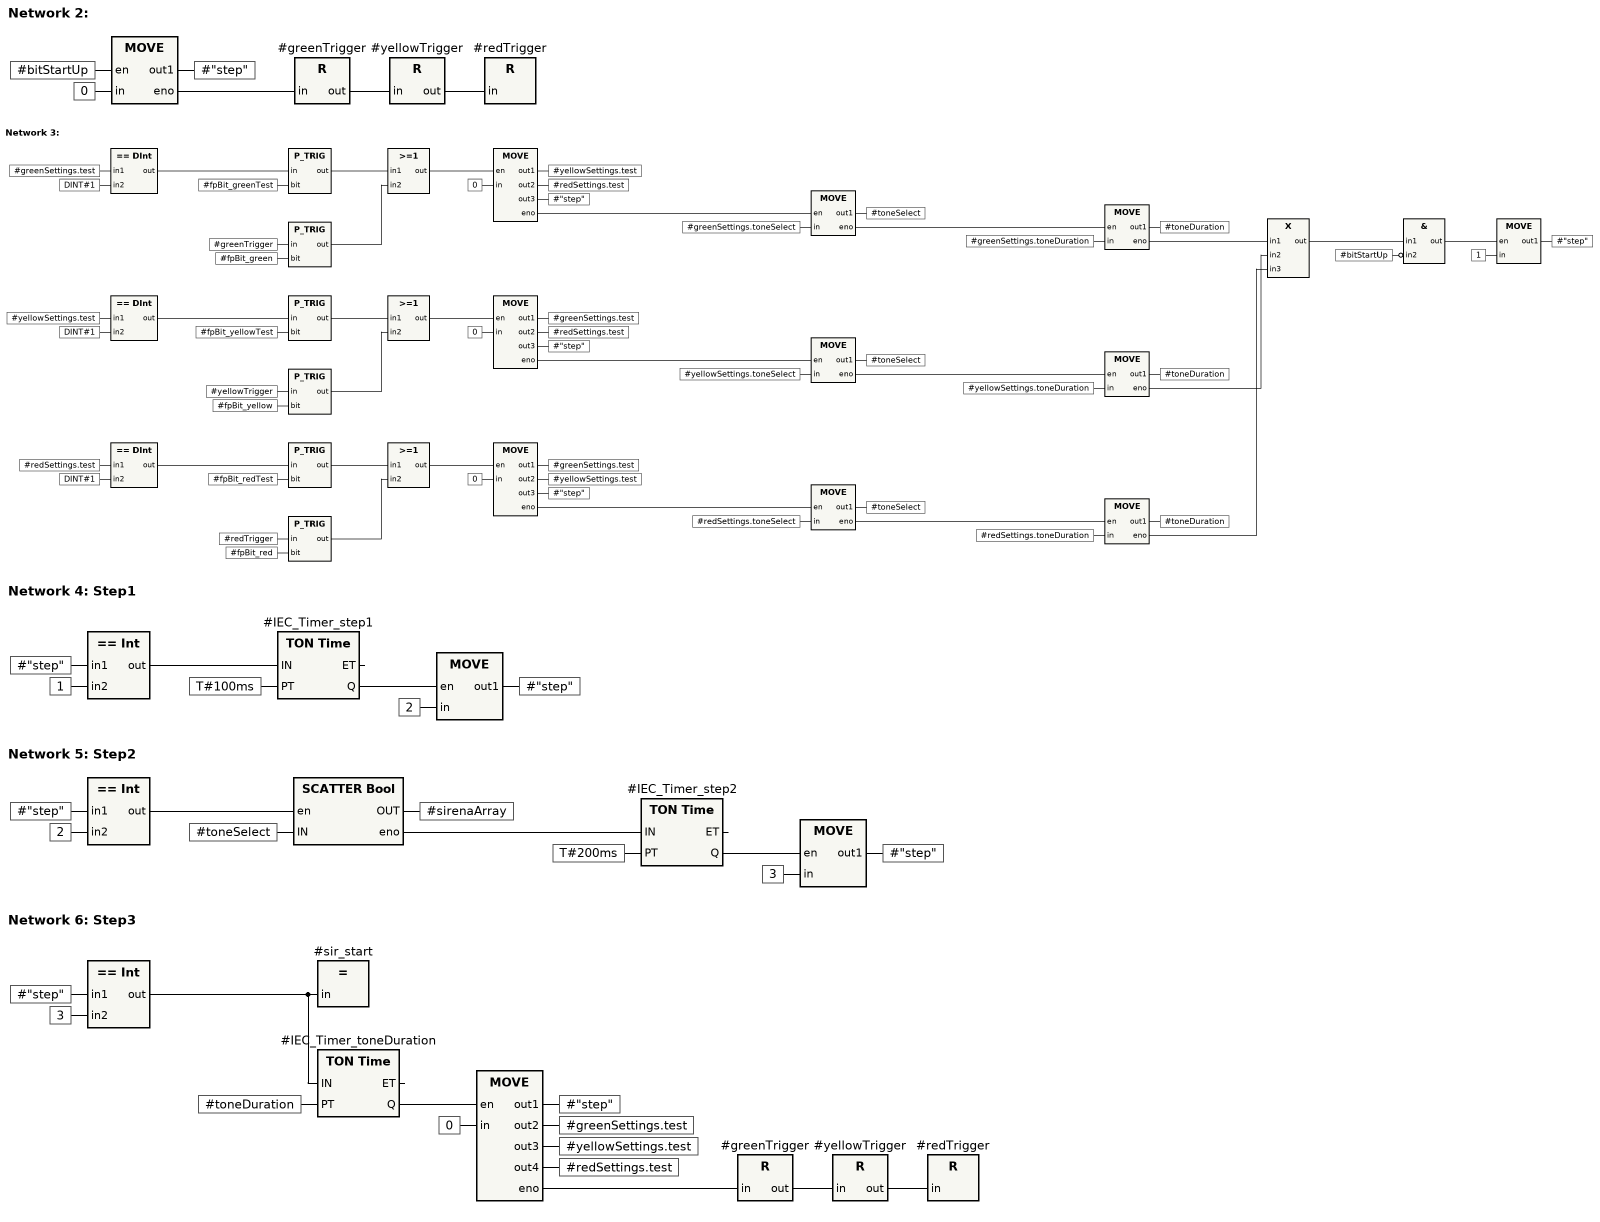
   IF #bitStartUp THEN
       #"step" := 0;
       #greenTrigger := FALSE;
       #yellowTrigger := FALSE;
       #redTrigger := FALSE;
   END_IF;
END_REGION

REGION Network 3
   #_w1 := #greenSettings.test = DINT#1;
   #_w2 := #_w1 AND NOT #fpBit_greenTest;   // rising edge
   #fpBit_greenTest := #_w1;
   #_w3 := #greenTrigger AND NOT #fpBit_green;   // rising edge
   #fpBit_green := #greenTrigger;
   #_w4 := #_w2 OR #_w3;
   IF #_w4 THEN
       #yellowSettings.test := 0;
       #redSettings.test := 0;
       #"step" := 0;
       #toneSelect := #greenSettings.toneSelect;
       #toneDuration := #greenSettings.toneDuration;
   END_IF;
   #_w5 := #yellowSettings.test = DINT#1;
   #_w6 := #_w5 AND NOT #fpBit_yellowTest;   // rising edge
   #fpBit_yellowTest := #_w5;
   #_w7 := #yellowTrigger AND NOT #fpBit_yellow;   // rising edge
   #fpBit_yellow := #yellowTrigger;
   #_w8 := #_w6 OR #_w7;
   IF #_w8 THEN
       #greenSettings.test := 0;
       #redSettings.test := 0;
       #"step" := 0;
       #toneSelect := #yellowSettings.toneSelect;
       #toneDuration := #yellowSettings.toneDuration;
   END_IF;
   #_w9 := #redSettings.test = DINT#1;
   #_w10 := #_w9 AND NOT #fpBit_redTest;   // rising edge
   #fpBit_redTest := #_w9;
   #_w11 := #redTrigger AND NOT #fpBit_red;   // rising edge
   #fpBit_red := #redTrigger;
   #_w12 := #_w10 OR #_w11;
   IF #_w12 THEN
       #greenSettings.test := 0;
       #yellowSettings.test := 0;
       #"step" := 0;
       #toneSelect := #redSettings.toneSelect;
       #toneDuration := #redSettings.toneDuration;
   END_IF;
   IF (#_w4 XOR #_w8 XOR #_w12) AND NOT #bitStartUp THEN #"step" := 1; END_IF;
END_REGION

REGION Network 4: Step1
   #IEC_Timer_step1.TON(IN := #"step" = 1, PT := T#100ms);
   IF #IEC_Timer_step1.Q THEN #"step" := 2; END_IF;
END_REGION

REGION Network 5: Step2
   #_w1 := #"step" = 2;
   SCATTER(EN := #_w1, IN := #toneSelect, OUT => #sirenaArray, ENO => #_w2);
   #IEC_Timer_step2.TON(IN := #_w2, PT := T#200ms);
   IF #IEC_Timer_step2.Q THEN #"step" := 3; END_IF;
END_REGION

REGION Network 6: Step3
   #sir_start := #"step" = 3;
   #IEC_Timer_toneDuration.TON(IN := #sir_start, PT := #toneDuration);
   IF #IEC_Timer_toneDuration.Q THEN
       #"step" := 0;
       #greenSettings.test := 0;
       #yellowSettings.test := 0;
       #redSettings.test := 0;
       #greenTrigger := FALSE;
       #yellowTrigger := FALSE;
       #redTrigger := FALSE;
   END_IF;
END_REGION

REGION Network 7: sirena_1
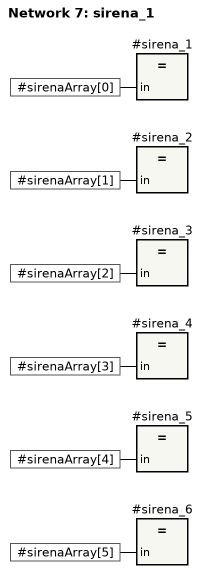
   #sirena_1 := #sirenaArray[0];
   #sirena_2 := #sirenaArray[1];
   #sirena_3 := #sirenaArray[2];
   #sirena_4 := #sirenaArray[3];
   #sirena_5 := #sirenaArray[4];
   #sirena_6 := #sirenaArray[5];
END_REGION
END_FUNCTION_BLOCK

FUNCTION_BLOCK "nokButtonMain"   // FB12, FBD
{ S7_Optimized_Access := 'TRUE' }
VERSION : 0.1
// stored: AutoNumber true, IsIECCheckEnabled false, IsRetainMemResEnabled false, MemoryReserve 100, SetENOAutomatically false, UDAEnableTagReadback false
   VAR
      nokButton1 { S7_SetPoint := 'True'} : "nokButton";
      nokButton2 { S7_SetPoint := 'True'} : "nokButton";
      nokButtonQUE_Instance { S7_SetPoint := 'True'} : "nokButtonQUE";
   END_VAR
BEGIN

REGION Network 1: NokButton1
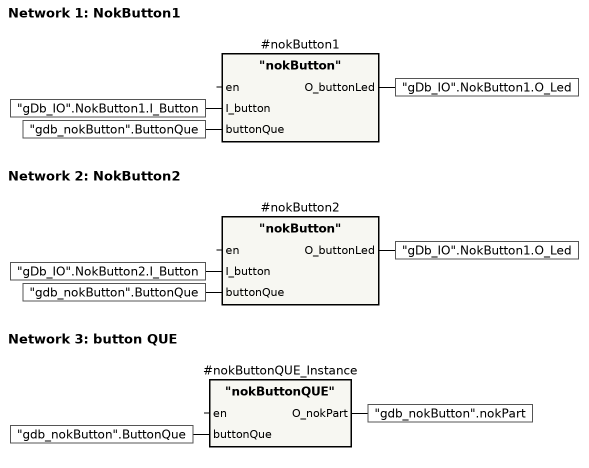
   #nokButton1(I_button := "gDb_IO".NokButton1.I_Button,   // "nokButton"
               buttonQue := "gdb_nokButton".ButtonQue,
               O_buttonLed => "gDb_IO".NokButton1.O_Led);
END_REGION

REGION Network 2: NokButton2
   #nokButton2(I_button := "gDb_IO".NokButton2.I_Button,   // "nokButton"
               buttonQue := "gdb_nokButton".ButtonQue,
               O_buttonLed => "gDb_IO".NokButton1.O_Led);
END_REGION

REGION Network 3: button QUE
   #nokButtonQUE_Instance(buttonQue := "gdb_nokButton".ButtonQue, O_nokPart => "gdb_nokButton".nokPart);   // "nokButtonQUE"
END_REGION
END_FUNCTION_BLOCK

FUNCTION_BLOCK "nokButton"   // FB11, FBD
{ S7_Optimized_Access := 'TRUE' }
VERSION : 0.1
// stored: AutoNumber true, IsIECCheckEnabled false, IsRetainMemResEnabled false, MemoryReserve 100, SetENOAutomatically false, UDAEnableTagReadback false
   VAR_INPUT
      I_button : Bool;
   END_VAR
   VAR_OUTPUT
      O_buttonLed : Bool;
   END_VAR
   VAR_IN_OUT
      buttonQue : Int;
   END_VAR
   VAR
      fpBit_button : Bool;
      SR_ButtonActive : Bool;
      fpBit_buttonActive : Bool;
      TO_Non_filter { S7_SetPoint := 'True'} : TON_TIME;
      buttonActive { ExternalAccessible := 'False'; ExternalVisible := 'False'; ExternalWritable := 'False'} : Bool;
   END_VAR
   VAR_TEMP
      fp_buttonActive : Bool;
   END_VAR
   VAR_TEMP   // added for the SCL form of the ladder/FBD networks
      _w1 : Bool;
      _w2 : Bool;
   END_VAR
BEGIN

REGION Network 2
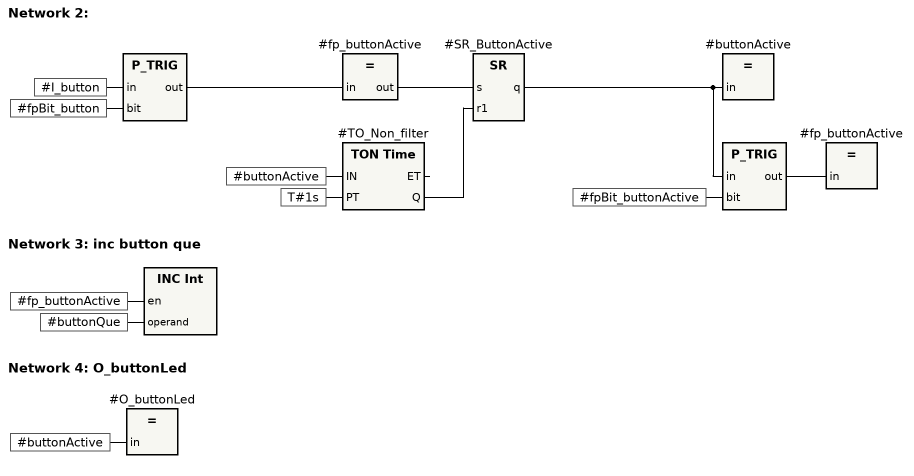
   #_w1 := #I_button AND NOT #fpBit_button;   // rising edge
   #fpBit_button := #I_button;
   #fp_buttonActive := #_w1;
   #TO_Non_filter(IN := #buttonActive, PT := T#1s);   // TON
   IF #_w1 THEN
       #SR_ButtonActive := TRUE;   // SR flip-flop
   END_IF;
   IF #TO_Non_filter.Q THEN #SR_ButtonActive := FALSE; END_IF;
   #buttonActive := #SR_ButtonActive;
   #_w2 := #SR_ButtonActive AND NOT #fpBit_buttonActive;   // rising edge
   #fpBit_buttonActive := #SR_ButtonActive;
   #fp_buttonActive := #_w2;
END_REGION

REGION Network 3: inc button que
   IF #fp_buttonActive THEN #buttonQue := #buttonQue + 1; END_IF;
END_REGION

REGION Network 4: O_buttonLed
   #O_buttonLed := #buttonActive;
END_REGION
END_FUNCTION_BLOCK

FUNCTION_BLOCK "nokButtonQUE"   // FB10, LAD
{ S7_Optimized_Access := 'TRUE' }
VERSION : 0.1
// stored: AutoNumber true, IsIECCheckEnabled false, IsRetainMemResEnabled false, MemoryReserve 100, SetENOAutomatically false, UDAEnableTagReadback false
   VAR_OUTPUT
      O_nokPart : Bool;
   END_VAR
   VAR_IN_OUT
      buttonQue : Int;
   END_VAR
   VAR
      "step" : Byte;
      TIM_countOn { S7_SetPoint := 'True'} : TON_TIME;
      TIM_countOff { S7_SetPoint := 'True'} : TON_TIME;
      countOn : Bool;
      countOff : Bool;
   END_VAR
BEGIN

REGION Network 1: Jump List
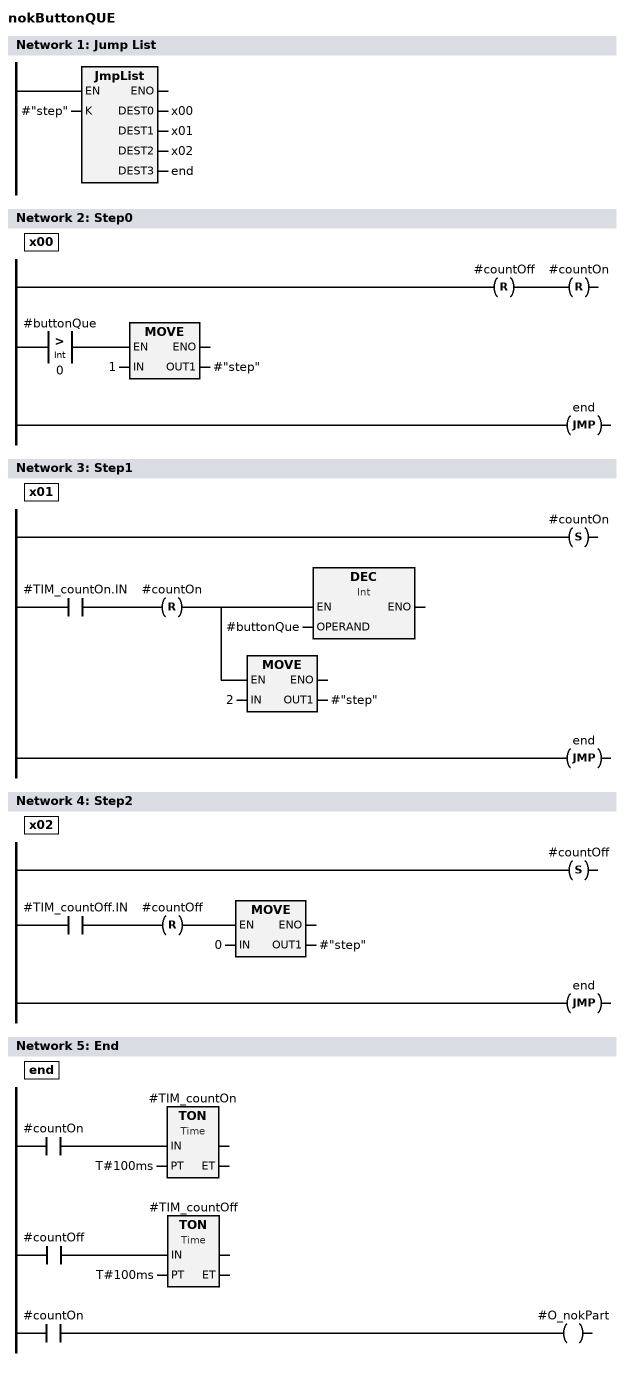
   // no SCL statement known for JmpList: written as a call
   JmpList(k := #"step", dest0 => x00, dest1 => x01, dest2 => x02, dest3 => end);
END_REGION

REGION Network 2: Step0
   Label( x00 )
   RUNG wire#powerrail
      R_Coil( #countOff )
      R_Coil( #countOn )
   END_RUNG
   RUNG wire#powerrail
      { S7_Templates := "SrcType := Int" } GT_Contact(in1 := #buttonQue, in2 := 0)
      Move(in := 1, out1 => #"step")
   END_RUNG
   RUNG wire#powerrail
      JumpCoil( end )
   END_RUNG
   // the same network as SCL:
   x00:
   #countOff := FALSE;
   #countOn := FALSE;
   IF #buttonQue > 0 THEN #"step" := 1; END_IF;
   GOTO end;
END_REGION

REGION Network 3: Step1
   Label( x01 )
   RUNG wire#powerrail
      S_Coil( #countOn )
   END_RUNG
   RUNG wire#powerrail
      Contact( #TIM_countOn.IN )
      R_Coil( #countOn )
      wire#w1
      { S7_Templates := "DestType := Int" } Dec( #buttonQue )
   END_RUNG
   RUNG wire#w1
      Move(in := 2, out1 => #"step")
   END_RUNG
   RUNG wire#powerrail
      JumpCoil( end )
   END_RUNG
   // the same network as SCL:
   x01:
   #countOn := TRUE;
   IF #TIM_countOn.IN THEN
       #countOn := FALSE;
       #buttonQue := #buttonQue - 1;
       #"step" := 2;
   END_IF;
   GOTO end;
END_REGION

REGION Network 4: Step2
   Label( x02 )
   RUNG wire#powerrail
      S_Coil( #countOff )
   END_RUNG
   RUNG wire#powerrail
      Contact( #TIM_countOff.IN )
      R_Coil( #countOff )
      Move(in := 0, out1 => #"step")
   END_RUNG
   RUNG wire#powerrail
      JumpCoil( end )
   END_RUNG
   // the same network as SCL:
   x02:
   #countOff := TRUE;
   IF #TIM_countOff.IN THEN
       #countOff := FALSE;
       #"step" := 0;
   END_IF;
   GOTO end;
END_REGION

REGION Network 5: End
   Label( end )
   RUNG wire#powerrail
      Contact( #countOn )
      { S7_Templates := "time_type := Time" } #TIM_countOn.TON(pt := T#100ms, et =>)
   END_RUNG
   RUNG wire#powerrail
      Contact( #countOff )
      { S7_Templates := "time_type := Time" } #TIM_countOff.TON(pt := T#100ms, et =>)
   END_RUNG
   RUNG wire#powerrail
      Contact( #countOn )
      Coil( #O_nokPart )
   END_RUNG
   // the same network as SCL:
   end:
   #TIM_countOn(IN := #countOn, PT := T#100ms);   // TON
   #TIM_countOff(IN := #countOff, PT := T#100ms);   // TON
   #O_nokPart := #countOn;
END_REGION
END_FUNCTION_BLOCK

FUNCTION_BLOCK "productionCounter"   // FB8, FBD
{ S7_Optimized_Access := 'TRUE' }
// stored: MemoryReserve 100, SetENOAutomatically false
   VAR_INPUT
      I_partProduced : Bool;
      I_nokPart : Bool;
   END_VAR
   VAR_IN_OUT
      IO_actualValues : "UDT_actualValues";
      IO_PreviousValues : "UDT_actualValues";
      IO_settings : "UDT_settings";
      IO_control : "UDT_control";
      IO_settingsShift1 : "UDT_settingsShift";
      IO_settingsShift2 : "UDT_settingsShift";
      IO_settingsShift3 : "UDT_settingsShift";
      IO_locTime : DTL;
   END_VAR
   VAR
      fpBit_resetCounters : Bool;
      fpBit_partProduced : Bool;
      fpBit_nokPart : Bool;
      fpBit_stop : Bool;
      fpBit_start : Bool;
      RS_taktTimeEn : Bool;
      TIM_taktTime { S7_SetPoint := 'True'} : TONR_TIME;
      memTaktTime : DInt;
      shiftTrigger0 { S7_SetPoint := 'True'} : "shiftTrigger";
      shiftTrigger1 { S7_SetPoint := 'True'} : "shiftTrigger";
      shiftTrigger2 { S7_SetPoint := 'True'} : "shiftTrigger";
      TaktTimeElapsed { S7_SetPoint := 'True'} : Time;
   END_VAR
   VAR_TEMP
      T_resetTaktTimeTimer : Bool;
      T_changeTaktTimeTimer : Bool;
      T_actualTOD : Time_Of_Day;
      T_shiftTrigger : Array[0..2] of Struct
         active : Bool;
         taktTimeEn : Bool;
         startDetect : Bool;
      END_STRUCT;
      T_control : Struct
         stop : Bool;
         start : Bool;
         resetCounters : Bool;
         taktTimeEn : Bool;
      END_STRUCT;
      T_settings : Struct
         enabled : Bool;
         autostartEnabled : Bool;
      END_STRUCT;
   END_VAR
   VAR_TEMP   // added for the SCL form of the ladder/FBD networks
      _w1 : Bool;
   END_VAR
BEGIN

REGION Network 1: free
END_REGION

REGION Network 2: actual TOD / Convert actual local time to TOD
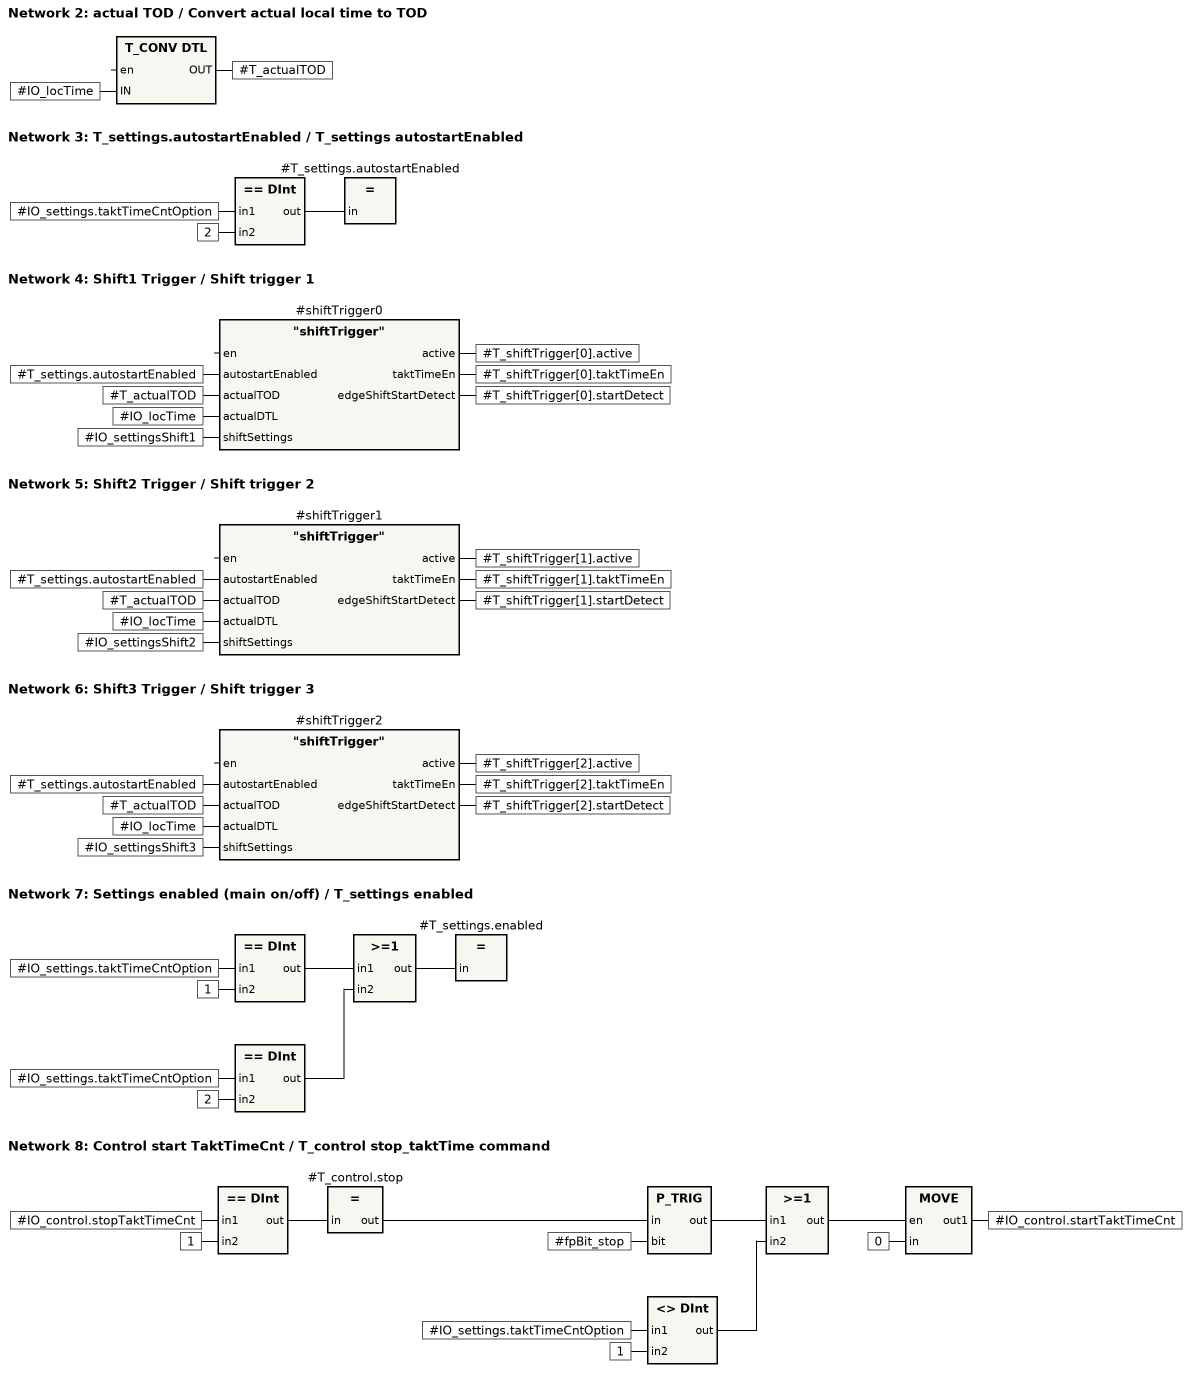
   T_CONV(IN := #IO_locTime, OUT => #T_actualTOD);
END_REGION

REGION Network 3: T_settings.autostartEnabled / T_settings autostartEnabled
   #T_settings.autostartEnabled := #IO_settings.taktTimeCntOption = 2;
END_REGION

REGION Network 4: Shift1 Trigger / Shift trigger 1
   #shiftTrigger0(autostartEnabled := #T_settings.autostartEnabled,   // "shiftTrigger"
                  actualTOD := #T_actualTOD,
                  actualDTL := #IO_locTime,
                  shiftSettings := #IO_settingsShift1,
                  active => #T_shiftTrigger[0].active,
                  taktTimeEn => #T_shiftTrigger[0].taktTimeEn,
                  edgeShiftStartDetect => #T_shiftTrigger[0].startDetect);
END_REGION

REGION Network 5: Shift2 Trigger / Shift trigger 2
   #shiftTrigger1(autostartEnabled := #T_settings.autostartEnabled,   // "shiftTrigger"
                  actualTOD := #T_actualTOD,
                  actualDTL := #IO_locTime,
                  shiftSettings := #IO_settingsShift2,
                  active => #T_shiftTrigger[1].active,
                  taktTimeEn => #T_shiftTrigger[1].taktTimeEn,
                  edgeShiftStartDetect => #T_shiftTrigger[1].startDetect);
END_REGION

REGION Network 6: Shift3 Trigger / Shift trigger 3
   #shiftTrigger2(autostartEnabled := #T_settings.autostartEnabled,   // "shiftTrigger"
                  actualTOD := #T_actualTOD,
                  actualDTL := #IO_locTime,
                  shiftSettings := #IO_settingsShift3,
                  active => #T_shiftTrigger[2].active,
                  taktTimeEn => #T_shiftTrigger[2].taktTimeEn,
                  edgeShiftStartDetect => #T_shiftTrigger[2].startDetect);
END_REGION

REGION Network 7: Settings enabled (main on/off) / T_settings enabled
   #T_settings.enabled := (#IO_settings.taktTimeCntOption = 1) OR (#IO_settings.taktTimeCntOption = 2);
END_REGION

REGION Network 8: Control start TaktTimeCnt / T_control stop_taktTime command
   #T_control.stop := #IO_control.stopTaktTimeCnt = 1;
   #_w1 := #T_control.stop AND NOT #fpBit_stop;   // rising edge
   #fpBit_stop := #T_control.stop;
   IF #_w1 OR (#IO_settings.taktTimeCntOption <> 1) THEN #IO_control.startTaktTimeCnt := 0; END_IF;
END_REGION

REGION Network 9: Control stop TaktTimeCnt / T_control start_taktTime command
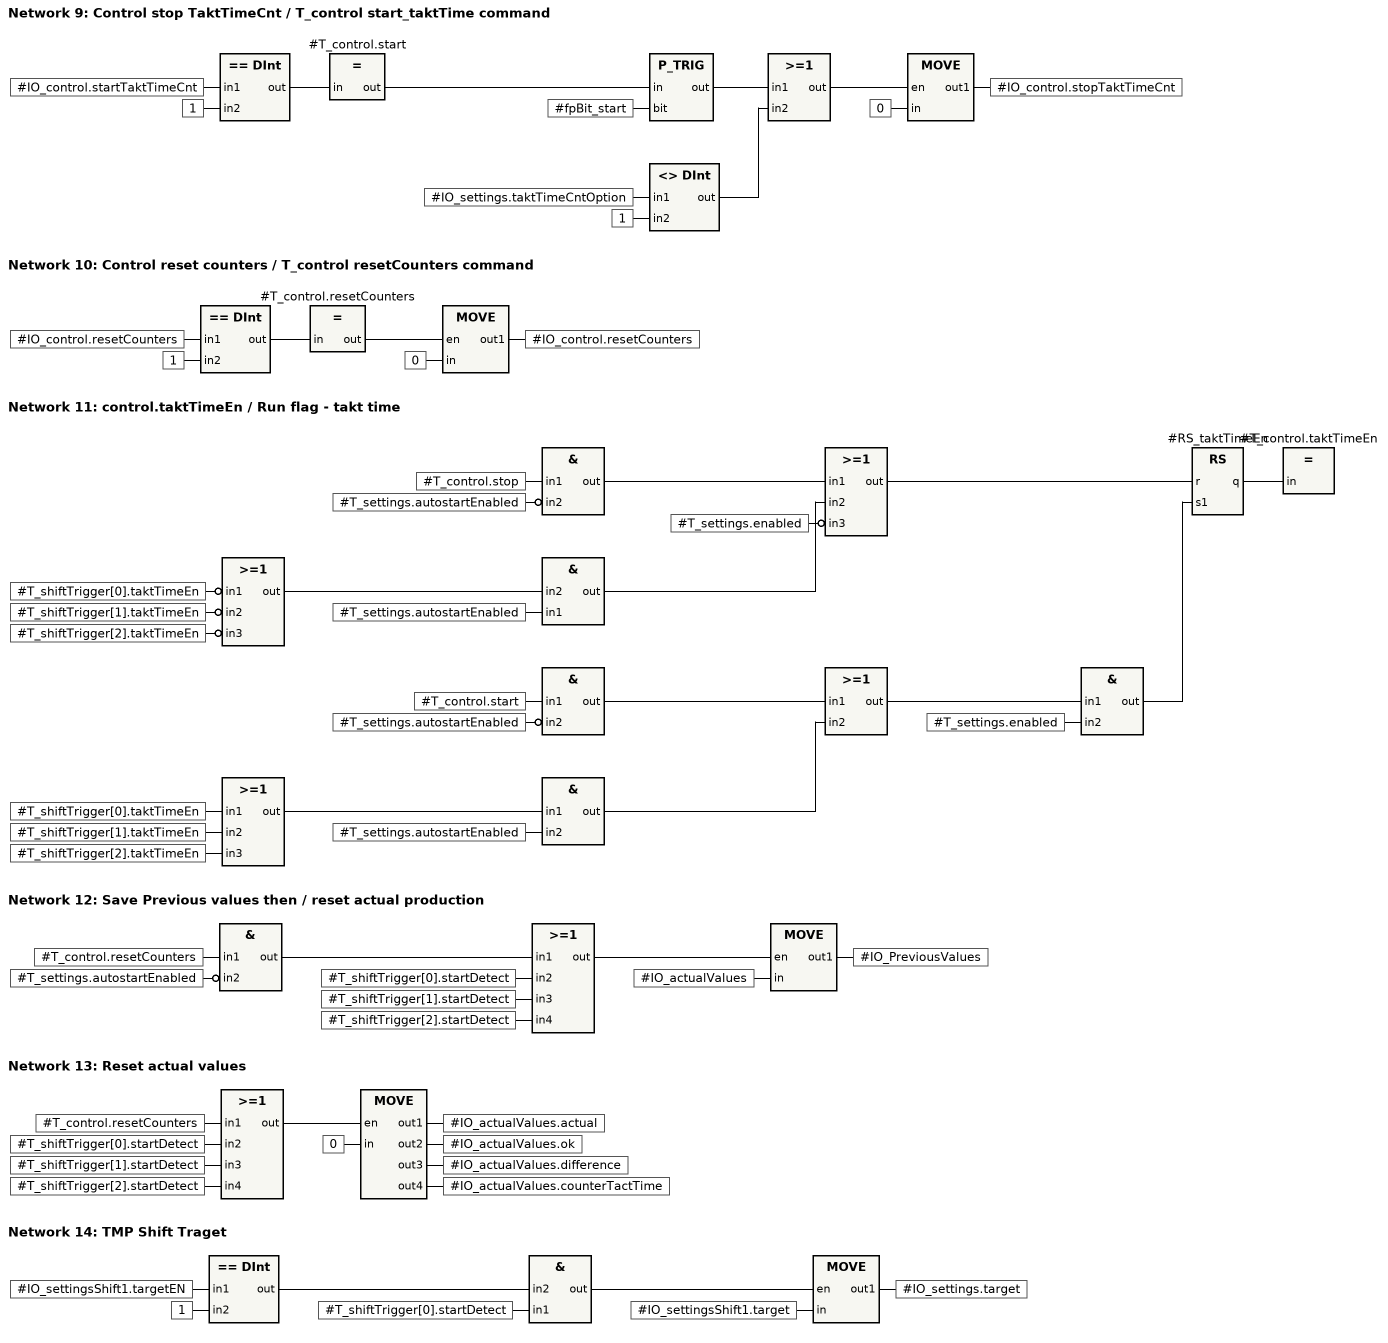
   #T_control.start := #IO_control.startTaktTimeCnt = 1;
   #_w1 := #T_control.start AND NOT #fpBit_start;   // rising edge
   #fpBit_start := #T_control.start;
   IF #_w1 OR (#IO_settings.taktTimeCntOption <> 1) THEN #IO_control.stopTaktTimeCnt := 0; END_IF;
END_REGION

REGION Network 10: Control reset counters / T_control resetCounters command
   #T_control.resetCounters := #IO_control.resetCounters = 1;
   IF #T_control.resetCounters THEN #IO_control.resetCounters := 0; END_IF;
END_REGION

REGION Network 11: control.taktTimeEn / Run flag - takt time
   IF (#T_control.stop AND NOT #T_settings.autostartEnabled) OR ((NOT #T_shiftTrigger[0].taktTimeEn OR NOT #T_shiftTrigger[1].taktTimeEn OR NOT #T_shiftTrigger[2].taktTimeEn) AND #T_settings.autostartEnabled) OR NOT #T_settings.enabled THEN
       #RS_taktTimeEn := FALSE;   // RS flip-flop
   END_IF;
   IF ((#T_control.start AND NOT #T_settings.autostartEnabled) OR ((#T_shiftTrigger[0].taktTimeEn OR #T_shiftTrigger[1].taktTimeEn OR #T_shiftTrigger[2].taktTimeEn) AND #T_settings.autostartEnabled)) AND #T_settings.enabled THEN
       #RS_taktTimeEn := TRUE;
   END_IF;
   #T_control.taktTimeEn := #RS_taktTimeEn;
END_REGION

REGION Network 12: Save Previous values then / reset actual production
   IF (#T_control.resetCounters AND NOT #T_settings.autostartEnabled) OR #T_shiftTrigger[0].startDetect OR #T_shiftTrigger[1].startDetect OR #T_shiftTrigger[2].startDetect THEN
       #IO_PreviousValues := #IO_actualValues;
   END_IF;
END_REGION

REGION Network 13: Reset actual values
   IF #T_control.resetCounters OR #T_shiftTrigger[0].startDetect OR #T_shiftTrigger[1].startDetect OR #T_shiftTrigger[2].startDetect THEN
       #IO_actualValues.actual := 0;
       #IO_actualValues.ok := 0;
       #IO_actualValues.difference := 0;
       #IO_actualValues.counterTactTime := 0;
   END_IF;
END_REGION

REGION Network 14: TMP Shift Traget
   IF (#IO_settingsShift1.targetEN = 1) AND #T_shiftTrigger[0].startDetect THEN
       #IO_settings.target := #IO_settingsShift1.target;
   END_IF;
END_REGION

REGION Network 15: #IO_settingsShift1.target - > #IO_settings.target
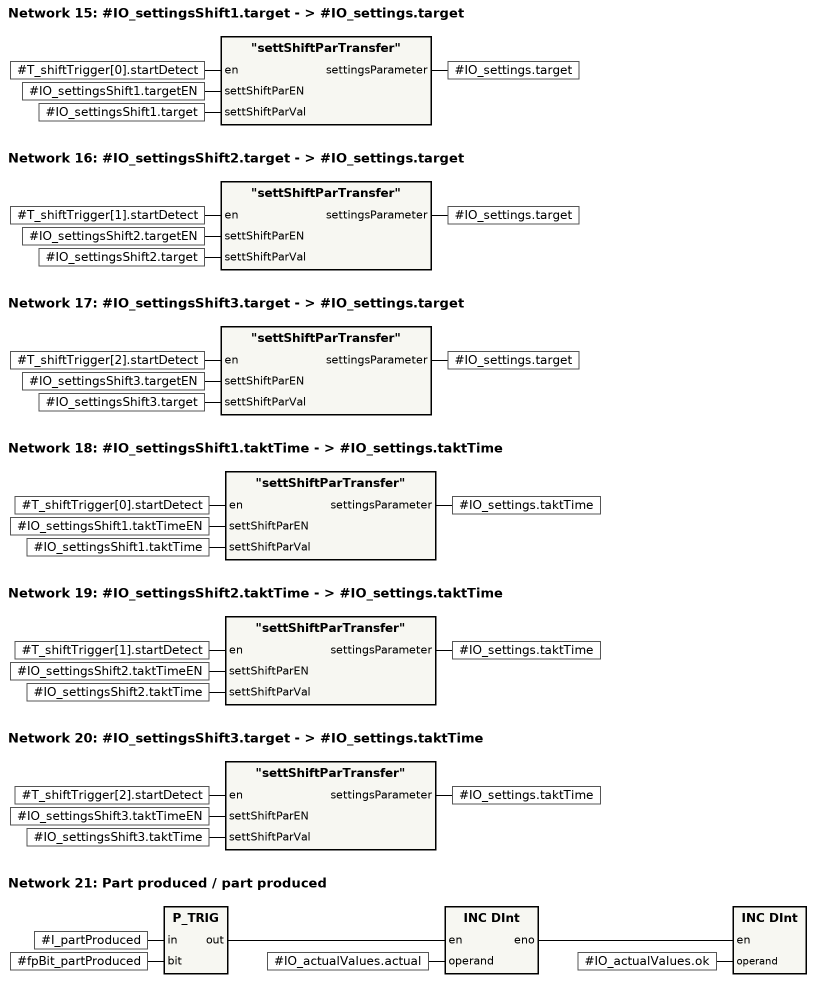
   IF #T_shiftTrigger[0].startDetect THEN
       "settShiftParTransfer"(settShiftParEN := #IO_settingsShift1.targetEN,
                              settShiftParVal := #IO_settingsShift1.target,
                              settingsParameter => #IO_settings.target);
   END_IF;
END_REGION

REGION Network 16: #IO_settingsShift2.target - > #IO_settings.target
   IF #T_shiftTrigger[1].startDetect THEN
       "settShiftParTransfer"(settShiftParEN := #IO_settingsShift2.targetEN,
                              settShiftParVal := #IO_settingsShift2.target,
                              settingsParameter => #IO_settings.target);
   END_IF;
END_REGION

REGION Network 17: #IO_settingsShift3.target - > #IO_settings.target
   IF #T_shiftTrigger[2].startDetect THEN
       "settShiftParTransfer"(settShiftParEN := #IO_settingsShift3.targetEN,
                              settShiftParVal := #IO_settingsShift3.target,
                              settingsParameter => #IO_settings.target);
   END_IF;
END_REGION

REGION Network 18: #IO_settingsShift1.taktTime - > #IO_settings.taktTime
   IF #T_shiftTrigger[0].startDetect THEN
       "settShiftParTransfer"(settShiftParEN := #IO_settingsShift1.taktTimeEN,
                              settShiftParVal := #IO_settingsShift1.taktTime,
                              settingsParameter => #IO_settings.taktTime);
   END_IF;
END_REGION

REGION Network 19: #IO_settingsShift2.taktTime - > #IO_settings.taktTime
   IF #T_shiftTrigger[1].startDetect THEN
       "settShiftParTransfer"(settShiftParEN := #IO_settingsShift2.taktTimeEN,
                              settShiftParVal := #IO_settingsShift2.taktTime,
                              settingsParameter => #IO_settings.taktTime);
   END_IF;
END_REGION

REGION Network 20: #IO_settingsShift3.target - > #IO_settings.taktTime
   IF #T_shiftTrigger[2].startDetect THEN
       "settShiftParTransfer"(settShiftParEN := #IO_settingsShift3.taktTimeEN,
                              settShiftParVal := #IO_settingsShift3.taktTime,
                              settingsParameter => #IO_settings.taktTime);
   END_IF;
END_REGION

REGION Network 21: Part produced / part produced
   // ENO of a box is taken as its EN; it also drops when the box reports an error
   #_w1 := #I_partProduced AND NOT #fpBit_partProduced;   // rising edge
   #fpBit_partProduced := #I_partProduced;
   IF #_w1 THEN
       #IO_actualValues.actual := #IO_actualValues.actual + 1;
       #IO_actualValues.ok := #IO_actualValues.ok + 1;
   END_IF;
END_REGION

REGION Network 22: Nok part / NOK part
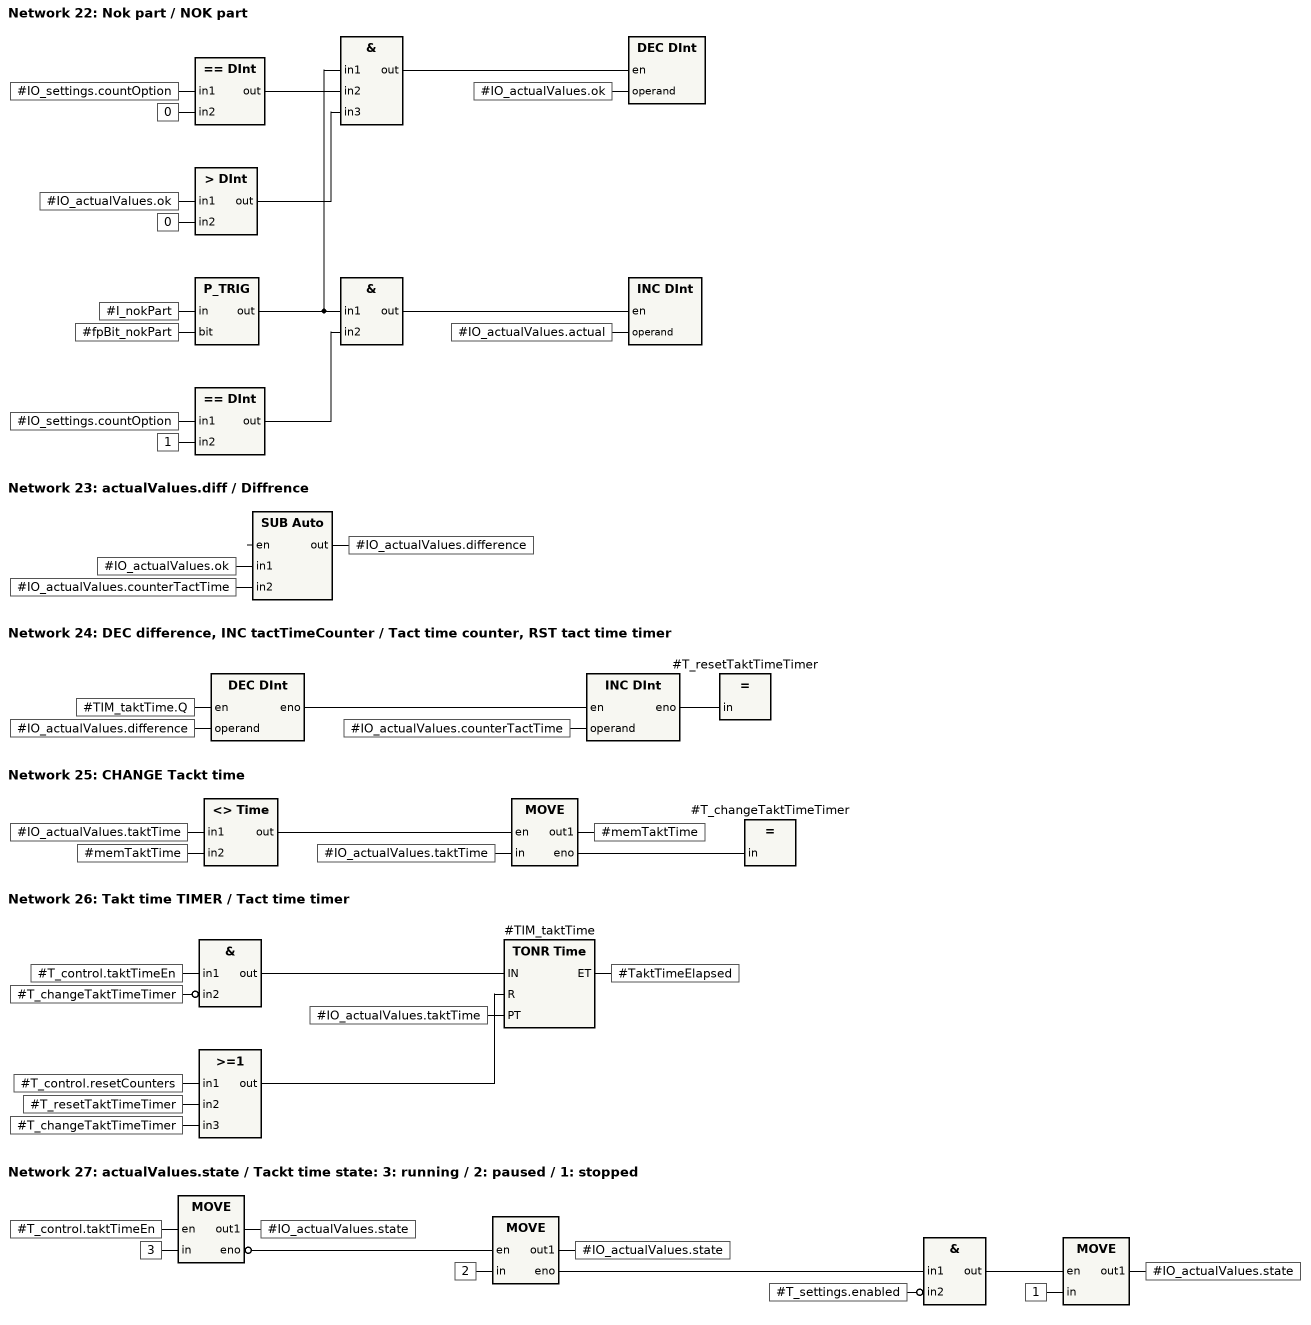
   #_w1 := #I_nokPart AND NOT #fpBit_nokPart;   // rising edge
   #fpBit_nokPart := #I_nokPart;
   IF #_w1 AND (#IO_settings.countOption = 0) AND (#IO_actualValues.ok > 0) THEN
       #IO_actualValues.ok := #IO_actualValues.ok - 1;
   END_IF;
   IF #_w1 AND (#IO_settings.countOption = 1) THEN
       #IO_actualValues.actual := #IO_actualValues.actual + 1;
   END_IF;
END_REGION

REGION Network 23: actualValues.diff / Diffrence
   #IO_actualValues.difference := #IO_actualValues.ok - #IO_actualValues.counterTactTime;
END_REGION

REGION Network 24: DEC difference, INC tactTimeCounter / Tact time counter, RST tact time timer
   // ENO of a box is taken as its EN; it also drops when the box reports an error
   IF #TIM_taktTime.Q THEN
       #IO_actualValues.difference := #IO_actualValues.difference - 1;
       #IO_actualValues.counterTactTime := #IO_actualValues.counterTactTime + 1;
   END_IF;
   #T_resetTaktTimeTimer := #TIM_taktTime.Q;
END_REGION

REGION Network 25: CHANGE Tackt time
   #_w1 := #IO_actualValues.taktTime <> #memTaktTime;
   IF #_w1 THEN #memTaktTime := #IO_actualValues.taktTime; END_IF;
   #T_changeTaktTimeTimer := #_w1;
END_REGION

REGION Network 26: Takt time TIMER / Tact time timer
   #TIM_taktTime(IN := #T_control.taktTimeEn AND NOT #T_changeTaktTimeTimer,   // TONR
                 R := #T_control.resetCounters OR #T_resetTaktTimeTimer OR #T_changeTaktTimeTimer,
                 PT := #IO_actualValues.taktTime,
                 ET => #TaktTimeElapsed);
END_REGION

REGION Network 27: actualValues.state / Tackt time state: 3: running / 2: paused / 1: stopped
   // ENO of a box is taken as its EN; it also drops when the box reports an error
   IF #T_control.taktTimeEn THEN #IO_actualValues.state := 3; END_IF;
   #_w1 := NOT #T_control.taktTimeEn;
   IF #_w1 THEN #IO_actualValues.state := 2; END_IF;
   IF #_w1 AND NOT #T_settings.enabled THEN #IO_actualValues.state := 1; END_IF;
END_REGION

REGION Network 28: settings.target -> actualValues.Target
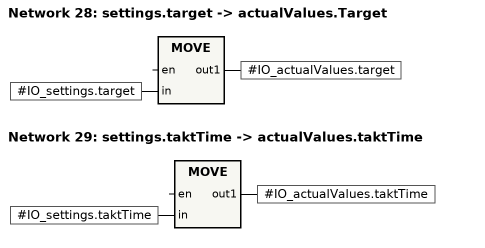
   #IO_actualValues.target := #IO_settings.target;
END_REGION

REGION Network 29: settings.taktTime -> actualValues.taktTime
   #IO_actualValues.taktTime := #IO_settings.taktTime;
END_REGION
END_FUNCTION_BLOCK

FUNCTION_BLOCK "shiftTrigger"   // FB4, FBD
{ S7_Optimized_Access := 'TRUE' }
// stored: MemoryReserve 100, SetENOAutomatically false
   VAR_INPUT
      autostartEnabled { ExternalAccessible := 'False'; ExternalVisible := 'False'; ExternalWritable := 'False'} : Bool;
      actualTOD { ExternalAccessible := 'False'; ExternalVisible := 'False'; ExternalWritable := 'False'} : Time_Of_Day;
      actualDTL : DTL;
      shiftSettings { ExternalAccessible := 'False'; ExternalVisible := 'False'; ExternalWritable := 'False'} : "UDT_settingsShift";
   END_VAR
   VAR_OUTPUT
      active : Bool;
      taktTimeEn { ExternalAccessible := 'False'; ExternalVisible := 'False'; ExternalWritable := 'False'} : Bool;
      edgeShiftStartDetect { ExternalAccessible := 'False'; ExternalVisible := 'False'; ExternalWritable := 'False'} : Bool;
   END_VAR
   VAR
      P_edgeShiftStartDetect : Bool;
   END_VAR
   VAR_TEMP
      T_shiftActive : Bool;
      T_break1Active : Bool;
      T_break2Active : Bool;
      T_break3Active : Bool;
      T_break4Active : Bool;
      T_break5Active : Bool;
      T_endShiftStartDetect : Time_Of_Day;
      T_ShiftStartDetect : Bool;
   END_VAR
   VAR_TEMP   // added for the SCL form of the ladder/FBD networks
      _w1 : Bool;
   END_VAR
BEGIN

REGION Network 1: Settings shift EN / Shift trigger disabled
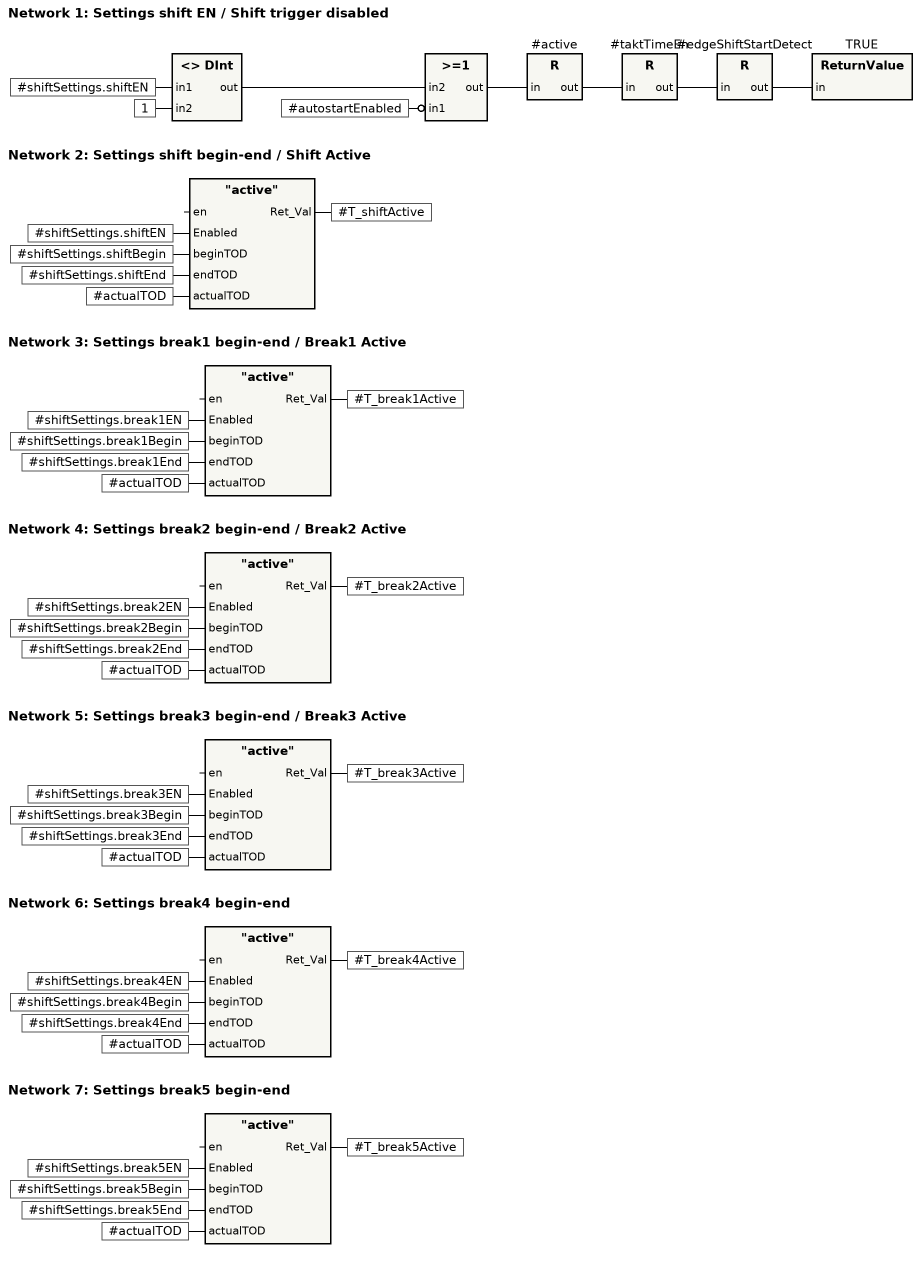
   #_w1 := (#shiftSettings.shiftEN <> 1) OR NOT #autostartEnabled;
   IF #_w1 THEN
       #active := FALSE;
       #taktTimeEn := FALSE;
       #edgeShiftStartDetect := FALSE;
       ENO := TRUE;
       RETURN;
   END_IF;
END_REGION

REGION Network 2: Settings shift begin-end / Shift Active
   #T_shiftActive := "active"(Enabled := #shiftSettings.shiftEN,
                           beginTOD := #shiftSettings.shiftBegin,
                           endTOD := #shiftSettings.shiftEnd,
                           actualTOD := #actualTOD);
END_REGION

REGION Network 3: Settings break1 begin-end / Break1 Active
   #T_break1Active := "active"(Enabled := #shiftSettings.break1EN,
                           beginTOD := #shiftSettings.break1Begin,
                           endTOD := #shiftSettings.break1End,
                           actualTOD := #actualTOD);
END_REGION

REGION Network 4: Settings break2 begin-end / Break2 Active
   #T_break2Active := "active"(Enabled := #shiftSettings.break2EN,
                           beginTOD := #shiftSettings.break2Begin,
                           endTOD := #shiftSettings.break2End,
                           actualTOD := #actualTOD);
END_REGION

REGION Network 5: Settings break3 begin-end / Break3 Active
   #T_break3Active := "active"(Enabled := #shiftSettings.break3EN,
                           beginTOD := #shiftSettings.break3Begin,
                           endTOD := #shiftSettings.break3End,
                           actualTOD := #actualTOD);
END_REGION

REGION Network 6: Settings break4 begin-end
   #T_break4Active := "active"(Enabled := #shiftSettings.break4EN,
                           beginTOD := #shiftSettings.break4Begin,
                           endTOD := #shiftSettings.break4End,
                           actualTOD := #actualTOD);
END_REGION

REGION Network 7: Settings break5 begin-end
   #T_break5Active := "active"(Enabled := #shiftSettings.break5EN,
                           beginTOD := #shiftSettings.break5Begin,
                           endTOD := #shiftSettings.break5End,
                           actualTOD := #actualTOD);
END_REGION

REGION Network 8: shift start detect signal duration
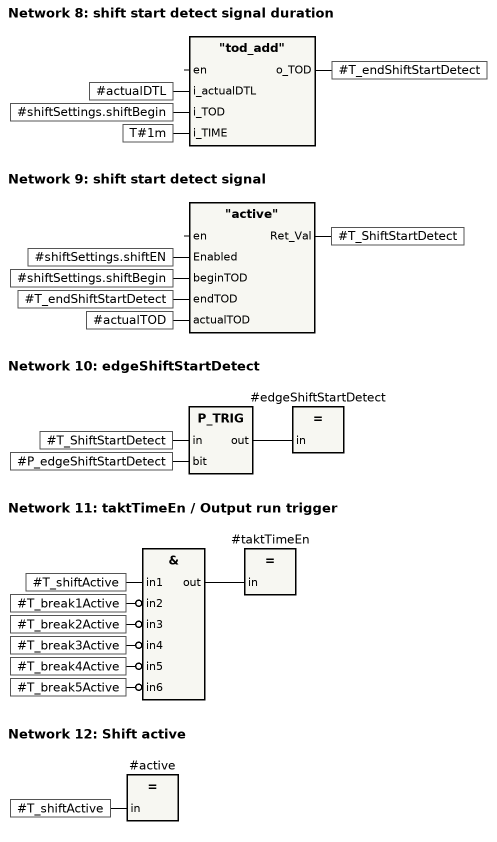
   "tod_add"(i_actualDTL := #actualDTL,
             i_TOD := #shiftSettings.shiftBegin,
             i_TIME := T#1m,
             o_TOD => #T_endShiftStartDetect);
END_REGION

REGION Network 9: shift start detect signal
   #T_ShiftStartDetect := "active"(Enabled := #shiftSettings.shiftEN,
                           beginTOD := #shiftSettings.shiftBegin,
                           endTOD := #T_endShiftStartDetect,
                           actualTOD := #actualTOD);
END_REGION

REGION Network 10: edgeShiftStartDetect
   #_w1 := #T_ShiftStartDetect AND NOT #P_edgeShiftStartDetect;   // rising edge
   #P_edgeShiftStartDetect := #T_ShiftStartDetect;
   #edgeShiftStartDetect := #_w1;
END_REGION

REGION Network 11: taktTimeEn / Output run trigger
   #taktTimeEn := #T_shiftActive AND NOT #T_break1Active AND NOT #T_break2Active AND NOT #T_break3Active AND NOT #T_break4Active AND NOT #T_break5Active;
END_REGION

REGION Network 12: Shift active
   #active := #T_shiftActive;
END_REGION
END_FUNCTION_BLOCK

FUNCTION "active" : Bool
{ S7_Optimized_Access := 'TRUE' }
VERSION : 0.1
   VAR_INPUT 
      Enabled : DInt;
      beginTOD : Time_Of_Day;
      endTOD : Time_Of_Day;
      actualTOD : Time_Of_Day;
   END_VAR

   VAR_TEMP 
      T_diff1 : Time;
      T_diff2 : Time;
   END_VAR


BEGIN
	#T_diff1 := "tod_diff"(endTOD := #endTOD, actual_begin_TOD := #actualTOD);
	#T_diff2 := "tod_diff"(endTOD := #endTOD, actual_begin_TOD := #beginTOD);
	
	IF #T_diff1 <= #T_diff2 AND #Enabled = 1 THEN
	    #active := TRUE;
	ELSE
	    #active := FALSE;
	END_IF;
	
	
	
	
	
	    
	    
END_FUNCTION

FUNCTION "tod_diff" : Time
{ S7_Optimized_Access := 'TRUE' }
VERSION : 0.1
   VAR_INPUT 
      endTOD : Time_Of_Day;
      actual_begin_TOD : Time_Of_Day;
   END_VAR


BEGIN
	#tod_diff := #endTOD - #actual_begin_TOD;
	IF #tod_diff < T#0ms THEN
	    #tod_diff := #tod_diff + T#24h;
	END_IF;
END_FUNCTION

FUNCTION "tod_add" : Void   // FC1, FBD
{ S7_Optimized_Access := 'TRUE' }
VERSION : 0.1
// stored: AutoNumber true, IsIECCheckEnabled false, SetENOAutomatically false, UDAEnableTagReadback false
   VAR_INPUT
      i_actualDTL : DTL;
      i_TOD : Time_Of_Day;
      i_TIME : Time;
   END_VAR
   VAR_OUTPUT
      o_TOD : Time_Of_Day;
   END_VAR
   VAR_TEMP
      tempDate : Date;
      tempDTL : DTL;
      tempDTL_1 : DTL;
   END_VAR
   VAR_TEMP   // added for the SCL form of the ladder/FBD networks
      _w1 : Bool;
      _w2 : Bool;
      _w3 : Bool;
   END_VAR
BEGIN

REGION Network 1: TOD add time(over midnight possible)
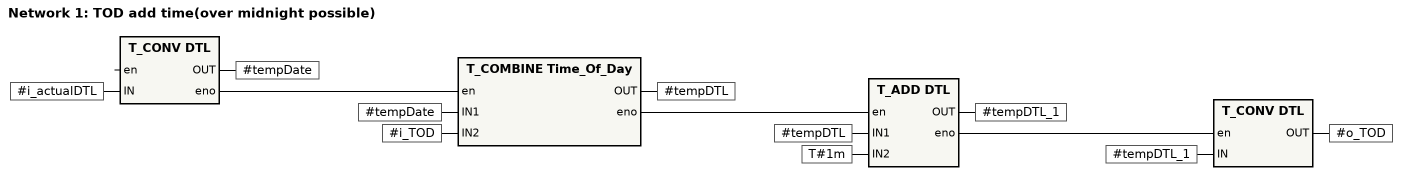
   T_CONV(IN := #i_actualDTL, OUT => #tempDate, ENO => #_w1);
   T_COMBINE(EN := #_w1, IN1 := #tempDate, IN2 := #i_TOD, OUT => #tempDTL, ENO => #_w2);
   T_ADD(EN := #_w2, IN1 := #tempDTL, IN2 := T#1m, OUT => #tempDTL_1, ENO => #_w3);
   IF #_w3 THEN T_CONV(IN := #tempDTL_1, OUT => #o_TOD); END_IF;
END_REGION
END_FUNCTION

FUNCTION "settShiftParTransfer" : Void   // FC5, FBD
{ S7_Optimized_Access := 'TRUE' }
// stored: SetENOAutomatically false
   VAR_INPUT
      settShiftParEN : DInt;
      settShiftParVal : DInt;
   END_VAR
   VAR_IN_OUT
      settingsParameter : DInt;
   END_VAR
BEGIN

REGION Network 1
